//     Term 27 (APS4322-7000)/Term 28 (APS4322-5000)/FB Inputs/H{1..9 step 2} Z-Field <-> Data Pointer/HallSensorFieldsXYZ[{107..119 step 3}]  (5 links)
//     Term 27 (APS4322-7000)/Term 28 (APS4322-5000)/FB Inputs/I{0..8 step 2} X-Field <-> Data Pointer/HallSensorFieldsXYZ[{120..132 step 3}]  (5 links)
//     Term 27 (APS4322-7000)/Term 28 (APS4322-5000)/FB Inputs/I{0..8 step 2} Y-Field <-> Data Pointer/HallSensorFieldsXYZ[{121..133 step 3}]  (5 links)
//     Term 27 (APS4322-7000)/Term 28 (APS4322-5000)/FB Inputs/I{0..8 step 2} Z-Field <-> Data Pointer/HallSensorFieldsXYZ[{122..134 step 3}]  (5 links)
//     Term 27 (APS4322-7000)/Term 28 (APS4322-5000)/FB Inputs/J{1..9 step 2} X-Field <-> Data Pointer/HallSensorFieldsXYZ[{135..147 step 3}]  (5 links)
//     Term 27 (APS4322-7000)/Term 28 (APS4322-5000)/FB Inputs/J{1..9 step 2} Y-Field <-> Data Pointer/HallSensorFieldsXYZ[{136..148 step 3}]  (5 links)
//     Term 27 (APS4322-7000)/Term 28 (APS4322-5000)/FB Inputs/J{1..9 step 2} Z-Field <-> Data Pointer/HallSensorFieldsXYZ[{137..149 step 3}]  (5 links)
//     Term 27 (APS4322-7000)/Term 28 (APS4322-5000)/FB Inputs/Status <-> Data Pointer/FeedbackStatus
//   Device 3 (EtherCAT) <-> TcCOM Objects/XPlanar/Part1/APS4322_P1_3
//     Term 17 (APS4322-7000)/APS Comm Inputs/CommStatusWord <-> Data Pointer/MoverCommStatusWord
//     Term 17 (APS4322-7000)/APS Comm Inputs/Data {1..4} <-> Data Pointer/MoverCommDataIn[{0..3}]  (4 links)
//     Term 17 (APS4322-7000)/APS Comm Outputs/CommControlWord <-> Data Pointer/MoverCommControlWord
//     Term 17 (APS4322-7000)/APS Comm Outputs/Data 1 <-> Data Pointer/MoverCommDataOut
//     Term 17 (APS4322-7000)/APS Diagdata/DC Link Voltage <-> Data Pointer/DcLinkVoltage
//     Term 17 (APS4322-7000)/APS Diagdata/Power supply current <-> Data Pointer/PowerSupplyCurrent
//     Term 17 (APS4322-7000)/APS Inputs/StatusWord <-> Data Pointer/PowerUnitStatusWord
//     Term 17 (APS4322-7000)/APS Outputs/ControlWord <-> Data Pointer/PowerUnitControlWord
//     Term 17 (APS4322-7000)/APS Outputs/Current D 0X0 <-> Data Pointer/DCurrentSetPoints[0]
//     Term 17 (APS4322-7000)/APS Outputs/Current D 0X1 <-> Data Pointer/DCurrentSetPoints[1]
//     Term 17 (APS4322-7000)/APS Outputs/Current D 0X2 <-> Data Pointer/DCurrentSetPoints[2]
//     Term 17 (APS4322-7000)/APS Outputs/Current D 1X0 <-> Data Pointer/DCurrentSetPoints[6]
//     Term 17 (APS4322-7000)/APS Outputs/Current D 1X1 <-> Data Pointer/DCurrentSetPoints[7]
//     Term 17 (APS4322-7000)/APS Outputs/Current D 1X2 <-> Data Pointer/DCurrentSetPoints[8]
//     Term 17 (APS4322-7000)/APS Outputs/Current D 2X0 <-> Data Pointer/DCurrentSetPoints[12]
//     Term 17 (APS4322-7000)/APS Outputs/Current D 2X1 <-> Data Pointer/DCurrentSetPoints[13]
//     Term 17 (APS4322-7000)/APS Outputs/Current D 2X2 <-> Data Pointer/DCurrentSetPoints[14]
//     Term 17 (APS4322-7000)/APS Outputs/Current D 3X0 <-> Data Pointer/DCurrentSetPoints[18]
//     Term 17 (APS4322-7000)/APS Outputs/Current D 3X1 <-> Data Pointer/DCurrentSetPoints[19]
//     Term 17 (APS4322-7000)/APS Outputs/Current D 3X2 <-> Data Pointer/DCurrentSetPoints[20]
//     Term 17 (APS4322-7000)/APS Outputs/Current D 0Y0 <-> Data Pointer/DCurrentSetPoints[3]
//     Term 17 (APS4322-7000)/APS Outputs/Current D 0Y1 <-> Data Pointer/DCurrentSetPoints[4]
//     Term 17 (APS4322-7000)/APS Outputs/Current D 0Y2 <-> Data Pointer/DCurrentSetPoints[5]
//     Term 17 (APS4322-7000)/APS Outputs/Current D 1Y0 <-> Data Pointer/DCurrentSetPoints[9]
//     Term 17 (APS4322-7000)/APS Outputs/Current D 1Y1 <-> Data Pointer/DCurrentSetPoints[10]
//     Term 17 (APS4322-7000)/APS Outputs/Current D 1Y2 <-> Data Pointer/DCurrentSetPoints[11]
//     Term 17 (APS4322-7000)/APS Outputs/Current D 2Y0 <-> Data Pointer/DCurrentSetPoints[15]
//     Term 17 (APS4322-7000)/APS Outputs/Current D 2Y1 <-> Data Pointer/DCurrentSetPoints[16]
//     Term 17 (APS4322-7000)/APS Outputs/Current D 2Y2 <-> Data Pointer/DCurrentSetPoints[17]
//     Term 17 (APS4322-7000)/APS Outputs/Current D 3Y0 <-> Data Pointer/DCurrentSetPoints[21]
//     Term 17 (APS4322-7000)/APS Outputs/Current D 3Y1 <-> Data Pointer/DCurrentSetPoints[22]
//     Term 17 (APS4322-7000)/APS Outputs/Current D 3Y2 <-> Data Pointer/DCurrentSetPoints[23]
//     Term 17 (APS4322-7000)/APS Outputs/Current Q 0X0 <-> Data Pointer/QCurrentSetPoints[0]
//     Term 17 (APS4322-7000)/APS Outputs/Current Q 0X1 <-> Data Pointer/QCurrentSetPoints[1]
//     Term 17 (APS4322-7000)/APS Outputs/Current Q 0X2 <-> Data Pointer/QCurrentSetPoints[2]
//     Term 17 (APS4322-7000)/APS Outputs/Current Q 1X0 <-> Data Pointer/QCurrentSetPoints[6]
//     Term 17 (APS4322-7000)/APS Outputs/Current Q 1X1 <-> Data Pointer/QCurrentSetPoints[7]
//     Term 17 (APS4322-7000)/APS Outputs/Current Q 1X2 <-> Data Pointer/QCurrentSetPoints[8]
//     Term 17 (APS4322-7000)/APS Outputs/Current Q 2X0 <-> Data Pointer/QCurrentSetPoints[12]
//     Term 17 (APS4322-7000)/APS Outputs/Current Q 2X1 <-> Data Pointer/QCurrentSetPoints[13]
//     Term 17 (APS4322-7000)/APS Outputs/Current Q 2X2 <-> Data Pointer/QCurrentSetPoints[14]
//     Term 17 (APS4322-7000)/APS Outputs/Current Q 3X0 <-> Data Pointer/QCurrentSetPoints[18]
//     Term 17 (APS4322-7000)/APS Outputs/Current Q 3X1 <-> Data Pointer/QCurrentSetPoints[19]
//     Term 17 (APS4322-7000)/APS Outputs/Current Q 3X2 <-> Data Pointer/QCurrentSetPoints[20]
//     Term 17 (APS4322-7000)/APS Outputs/Current Q 0Y0 <-> Data Pointer/QCurrentSetPoints[3]
//     Term 17 (APS4322-7000)/APS Outputs/Current Q 0Y1 <-> Data Pointer/QCurrentSetPoints[4]
//     Term 17 (APS4322-7000)/APS Outputs/Current Q 0Y2 <-> Data Pointer/QCurrentSetPoints[5]
//     Term 17 (APS4322-7000)/APS Outputs/Current Q 1Y0 <-> Data Pointer/QCurrentSetPoints[9]
//     Term 17 (APS4322-7000)/APS Outputs/Current Q 1Y1 <-> Data Pointer/QCurrentSetPoints[10]
//     Term 17 (APS4322-7000)/APS Outputs/Current Q 1Y2 <-> Data Pointer/QCurrentSetPoints[11]
//     Term 17 (APS4322-7000)/APS Outputs/Current Q 2Y0 <-> Data Pointer/QCurrentSetPoints[15]
//     Term 17 (APS4322-7000)/APS Outputs/Current Q 2Y1 <-> Data Pointer/QCurrentSetPoints[16]
//     Term 17 (APS4322-7000)/APS Outputs/Current Q 2Y2 <-> Data Pointer/QCurrentSetPoints[17]
//     Term 17 (APS4322-7000)/APS Outputs/Current Q 3Y0 <-> Data Pointer/QCurrentSetPoints[21]
//     Term 17 (APS4322-7000)/APS Outputs/Current Q 3Y1 <-> Data Pointer/QCurrentSetPoints[22]
//     Term 17 (APS4322-7000)/APS Outputs/Current Q 3Y2 <-> Data Pointer/QCurrentSetPoints[23]
//     Term 17 (APS4322-7000)/APS Outputs/PhiE 0X0 <-> Data Pointer/PhiSetPoints[0]
//     Term 17 (APS4322-7000)/APS Outputs/PhiE 0X1 <-> Data Pointer/PhiSetPoints[1]
//     Term 17 (APS4322-7000)/APS Outputs/PhiE 0X2 <-> Data Pointer/PhiSetPoints[2]
//     Term 17 (APS4322-7000)/APS Outputs/PhiE 1X0 <-> Data Pointer/PhiSetPoints[6]
//     Term 17 (APS4322-7000)/APS Outputs/PhiE 1X1 <-> Data Pointer/PhiSetPoints[7]
//     Term 17 (APS4322-7000)/APS Outputs/PhiE 1X2 <-> Data Pointer/PhiSetPoints[8]
//     Term 17 (APS4322-7000)/APS Outputs/PhiE 2X0 <-> Data Pointer/PhiSetPoints[12]
//     Term 17 (APS4322-7000)/APS Outputs/PhiE 2X1 <-> Data Pointer/PhiSetPoints[13]
//     Term 17 (APS4322-7000)/APS Outputs/PhiE 2X2 <-> Data Pointer/PhiSetPoints[14]
//     Term 17 (APS4322-7000)/APS Outputs/PhiE 3X0 <-> Data Pointer/PhiSetPoints[18]
//     Term 17 (APS4322-7000)/APS Outputs/PhiE 3X1 <-> Data Pointer/PhiSetPoints[19]
//     Term 17 (APS4322-7000)/APS Outputs/PhiE 3X2 <-> Data Pointer/PhiSetPoints[20]
//     Term 17 (APS4322-7000)/APS Outputs/PhiE 0Y0 <-> Data Pointer/PhiSetPoints[3]
//     Term 17 (APS4322-7000)/APS Outputs/PhiE 0Y1 <-> Data Pointer/PhiSetPoints[4]
//     Term 17 (APS4322-7000)/APS Outputs/PhiE 0Y2 <-> Data Pointer/PhiSetPoints[5]
//     Term 17 (APS4322-7000)/APS Outputs/PhiE 1Y0 <-> Data Pointer/PhiSetPoints[9]
//     Term 17 (APS4322-7000)/APS Outputs/PhiE 1Y1 <-> Data Pointer/PhiSetPoints[10]
//     Term 17 (APS4322-7000)/APS Outputs/PhiE 1Y2 <-> Data Pointer/PhiSetPoints[11]
//     Term 17 (APS4322-7000)/APS Outputs/PhiE 2Y0 <-> Data Pointer/PhiSetPoints[15]
//     Term 17 (APS4322-7000)/APS Outputs/PhiE 2Y1 <-> Data Pointer/PhiSetPoints[16]
//     Term 17 (APS4322-7000)/APS Outputs/PhiE 2Y2 <-> Data Pointer/PhiSetPoints[17]
//     Term 17 (APS4322-7000)/APS Outputs/PhiE 3Y0 <-> Data Pointer/PhiSetPoints[21]
//     Term 17 (APS4322-7000)/APS Outputs/PhiE 3Y1 <-> Data Pointer/PhiSetPoints[22]
//     Term 17 (APS4322-7000)/APS Outputs/PhiE 3Y2 <-> Data Pointer/PhiSetPoints[23]
//     Term 17 (APS4322-7000)/Term 18 (APS4322-5000)/FB Inputs/A{0..8 step 2} X-Field <-> Data Pointer/HallSensorFieldsXYZ[{0..12 step 3}]  (5 links)
//     Term 17 (APS4322-7000)/Term 18 (APS4322-5000)/FB Inputs/A{0..8 step 2} Y-Field <-> Data Pointer/HallSensorFieldsXYZ[{1..13 step 3}]  (5 links)
//     Term 17 (APS4322-7000)/Term 18 (APS4322-5000)/FB Inputs/A{0..8 step 2} Z-Field <-> Data Pointer/HallSensorFieldsXYZ[{2..14 step 3}]  (5 links)
//     Term 17 (APS4322-7000)/Term 18 (APS4322-5000)/FB Inputs/B{1..9 step 2} X-Field <-> Data Pointer/HallSensorFieldsXYZ[{15..27 step 3}]  (5 links)
//     Term 17 (APS4322-7000)/Term 18 (APS4322-5000)/FB Inputs/B{1..9 step 2} Y-Field <-> Data Pointer/HallSensorFieldsXYZ[{16..28 step 3}]  (5 links)
//     Term 17 (APS4322-7000)/Term 18 (APS4322-5000)/FB Inputs/B{1..9 step 2} Z-Field <-> Data Pointer/HallSensorFieldsXYZ[{17..29 step 3}]  (5 links)
//     Term 17 (APS4322-7000)/Term 18 (APS4322-5000)/FB Inputs/C{0..8 step 2} X-Field <-> Data Pointer/HallSensorFieldsXYZ[{30..42 step 3}]  (5 links)
//     Term 17 (APS4322-7000)/Term 18 (APS4322-5000)/FB Inputs/C{0..8 step 2} Y-Field <-> Data Pointer/HallSensorFieldsXYZ[{31..43 step 3}]  (5 links)
//     Term 17 (APS4322-7000)/Term 18 (APS4322-5000)/FB Inputs/C{0..8 step 2} Z-Field <-> Data Pointer/HallSensorFieldsXYZ[{32..44 step 3}]  (5 links)
//     Term 17 (APS4322-7000)/Term 18 (APS4322-5000)/FB Inputs/D{1..9 step 2} X-Field <-> Data Pointer/HallSensorFieldsXYZ[{45..57 step 3}]  (5 links)
//     Term 17 (APS4322-7000)/Term 18 (APS4322-5000)/FB Inputs/D{1..9 step 2} Y-Field <-> Data Pointer/HallSensorFieldsXYZ[{46..58 step 3}]  (5 links)
//     Term 17 (APS4322-7000)/Term 18 (APS4322-5000)/FB Inputs/D{1..9 step 2} Z-Field <-> Data Pointer/HallSensorFieldsXYZ[{47..59 step 3}]  (5 links)
//     Term 17 (APS4322-7000)/Term 18 (APS4322-5000)/FB Inputs/E{0..8 step 2} X-Field <-> Data Pointer/HallSensorFieldsXYZ[{60..72 step 3}]  (5 links)
//     Term 17 (APS4322-7000)/Term 18 (APS4322-5000)/FB Inputs/E{0..8 step 2} Y-Field <-> Data Pointer/HallSensorFieldsXYZ[{61..73 step 3}]  (5 links)
//     Term 17 (APS4322-7000)/Term 18 (APS4322-5000)/FB Inputs/E{0..8 step 2} Z-Field <-> Data Pointer/HallSensorFieldsXYZ[{62..74 step 3}]  (5 links)
//     Term 17 (APS4322-7000)/Term 18 (APS4322-5000)/FB Inputs/F{1..9 step 2} X-Field <-> Data Pointer/HallSensorFieldsXYZ[{75..87 step 3}]  (5 links)
//     Term 17 (APS4322-7000)/Term 18 (APS4322-5000)/FB Inputs/F{1..9 step 2} Y-Field <-> Data Pointer/HallSensorFieldsXYZ[{76..88 step 3}]  (5 links)
//     Term 17 (APS4322-7000)/Term 18 (APS4322-5000)/FB Inputs/F{1..9 step 2} Z-Field <-> Data Pointer/HallSensorFieldsXYZ[{77..89 step 3}]  (5 links)
//     Term 17 (APS4322-7000)/Term 18 (APS4322-5000)/FB Inputs/G{0..8 step 2} X-Field <-> Data Pointer/HallSensorFieldsXYZ[{90..102 step 3}]  (5 links)
//     Term 17 (APS4322-7000)/Term 18 (APS4322-5000)/FB Inputs/G{0..8 step 2} Y-Field <-> Data Pointer/HallSensorFieldsXYZ[{91..103 step 3}]  (5 links)
//     Term 17 (APS4322-7000)/Term 18 (APS4322-5000)/FB Inputs/G{0..8 step 2} Z-Field <-> Data Pointer/HallSensorFieldsXYZ[{92..104 step 3}]  (5 links)
//     Term 17 (APS4322-7000)/Term 18 (APS4322-5000)/FB Inputs/H{1..9 step 2} X-Field <-> Data Pointer/HallSensorFieldsXYZ[{105..117 step 3}]  (5 links)
//     Term 17 (APS4322-7000)/Term 18 (APS4322-5000)/FB Inputs/H{1..9 step 2} Y-Field <-> Data Pointer/HallSensorFieldsXYZ[{106..118 step 3}]  (5 links)
//     Term 17 (APS4322-7000)/Term 18 (APS4322-5000)/FB Inputs/H{1..9 step 2} Z-Field <-> Data Pointer/HallSensorFieldsXYZ[{107..119 step 3}]  (5 links)
//     Term 17 (APS4322-7000)/Term 18 (APS4322-5000)/FB Inputs/I{0..8 step 2} X-Field <-> Data Pointer/HallSensorFieldsXYZ[{120..132 step 3}]  (5 links)
//     Term 17 (APS4322-7000)/Term 18 (APS4322-5000)/FB Inputs/I{0..8 step 2} Y-Field <-> Data Pointer/HallSensorFieldsXYZ[{121..133 step 3}]  (5 links)
//     Term 17 (APS4322-7000)/Term 18 (APS4322-5000)/FB Inputs/I{0..8 step 2} Z-Field <-> Data Pointer/HallSensorFieldsXYZ[{122..134 step 3}]  (5 links)
//     Term 17 (APS4322-7000)/Term 18 (APS4322-5000)/FB Inputs/J{1..9 step 2} X-Field <-> Data Pointer/HallSensorFieldsXYZ[{135..147 step 3}]  (5 links)
//     Term 17 (APS4322-7000)/Term 18 (APS4322-5000)/FB Inputs/J{1..9 step 2} Y-Field <-> Data Pointer/HallSensorFieldsXYZ[{136..148 step 3}]  (5 links)
//     Term 17 (APS4322-7000)/Term 18 (APS4322-5000)/FB Inputs/J{1..9 step 2} Z-Field <-> Data Pointer/HallSensorFieldsXYZ[{137..149 step 3}]  (5 links)
//     Term 17 (APS4322-7000)/Term 18 (APS4322-5000)/FB Inputs/Status <-> Data Pointer/FeedbackStatus
//   Device 3 (EtherCAT) <-> TcCOM Objects/XPlanar/Part1/APS4322_P1_4
//     Term 19 (APS4322-7000)/APS Comm Inputs/CommStatusWord <-> Data Pointer/MoverCommStatusWord
//     Term 19 (APS4322-7000)/APS Comm Inputs/Data {1..4} <-> Data Pointer/MoverCommDataIn[{0..3}]  (4 links)
//     Term 19 (APS4322-7000)/APS Comm Outputs/CommControlWord <-> Data Pointer/MoverCommControlWord
//     Term 19 (APS4322-7000)/APS Comm Outputs/Data 1 <-> Data Pointer/MoverCommDataOut
//     Term 19 (APS4322-7000)/APS Diagdata/DC Link Voltage <-> Data Pointer/DcLinkVoltage
//     Term 19 (APS4322-7000)/APS Diagdata/Power supply current <-> Data Pointer/PowerSupplyCurrent
//     Term 19 (APS4322-7000)/APS Inputs/StatusWord <-> Data Pointer/PowerUnitStatusWord
//     Term 19 (APS4322-7000)/APS Outputs/ControlWord <-> Data Pointer/PowerUnitControlWord
//     Term 19 (APS4322-7000)/APS Outputs/Current D 0X0 <-> Data Pointer/DCurrentSetPoints[0]
//     Term 19 (APS4322-7000)/APS Outputs/Current D 0X1 <-> Data Pointer/DCurrentSetPoints[1]
//     Term 19 (APS4322-7000)/APS Outputs/Current D 0X2 <-> Data Pointer/DCurrentSetPoints[2]
//     Term 19 (APS4322-7000)/APS Outputs/Current D 1X0 <-> Data Pointer/DCurrentSetPoints[6]
//     Term 19 (APS4322-7000)/APS Outputs/Current D 1X1 <-> Data Pointer/DCurrentSetPoints[7]
//     Term 19 (APS4322-7000)/APS Outputs/Current D 1X2 <-> Data Pointer/DCurrentSetPoints[8]
//     Term 19 (APS4322-7000)/APS Outputs/Current D 2X0 <-> Data Pointer/DCurrentSetPoints[12]
//     Term 19 (APS4322-7000)/APS Outputs/Current D 2X1 <-> Data Pointer/DCurrentSetPoints[13]
//     Term 19 (APS4322-7000)/APS Outputs/Current D 2X2 <-> Data Pointer/DCurrentSetPoints[14]
//     Term 19 (APS4322-7000)/APS Outputs/Current D 3X0 <-> Data Pointer/DCurrentSetPoints[18]
//     Term 19 (APS4322-7000)/APS Outputs/Current D 3X1 <-> Data Pointer/DCurrentSetPoints[19]
//     Term 19 (APS4322-7000)/APS Outputs/Current D 3X2 <-> Data Pointer/DCurrentSetPoints[20]
//     Term 19 (APS4322-7000)/APS Outputs/Current D 0Y0 <-> Data Pointer/DCurrentSetPoints[3]
//     Term 19 (APS4322-7000)/APS Outputs/Current D 0Y1 <-> Data Pointer/DCurrentSetPoints[4]
//     Term 19 (APS4322-7000)/APS Outputs/Current D 0Y2 <-> Data Pointer/DCurrentSetPoints[5]
//     Term 19 (APS4322-7000)/APS Outputs/Current D 1Y0 <-> Data Pointer/DCurrentSetPoints[9]
//     Term 19 (APS4322-7000)/APS Outputs/Current D 1Y1 <-> Data Pointer/DCurrentSetPoints[10]
//     Term 19 (APS4322-7000)/APS Outputs/Current D 1Y2 <-> Data Pointer/DCurrentSetPoints[11]
//     Term 19 (APS4322-7000)/APS Outputs/Current D 2Y0 <-> Data Pointer/DCurrentSetPoints[15]
//     Term 19 (APS4322-7000)/APS Outputs/Current D 2Y1 <-> Data Pointer/DCurrentSetPoints[16]
//     Term 19 (APS4322-7000)/APS Outputs/Current D 2Y2 <-> Data Pointer/DCurrentSetPoints[17]
//     Term 19 (APS4322-7000)/APS Outputs/Current D 3Y0 <-> Data Pointer/DCurrentSetPoints[21]
//     Term 19 (APS4322-7000)/APS Outputs/Current D 3Y1 <-> Data Pointer/DCurrentSetPoints[22]
//     Term 19 (APS4322-7000)/APS Outputs/Current D 3Y2 <-> Data Pointer/DCurrentSetPoints[23]
//     Term 19 (APS4322-7000)/APS Outputs/Current Q 0X0 <-> Data Pointer/QCurrentSetPoints[0]
//     Term 19 (APS4322-7000)/APS Outputs/Current Q 0X1 <-> Data Pointer/QCurrentSetPoints[1]
//     Term 19 (APS4322-7000)/APS Outputs/Current Q 0X2 <-> Data Pointer/QCurrentSetPoints[2]
//     Term 19 (APS4322-7000)/APS Outputs/Current Q 1X0 <-> Data Pointer/QCurrentSetPoints[6]
//     Term 19 (APS4322-7000)/APS Outputs/Current Q 1X1 <-> Data Pointer/QCurrentSetPoints[7]
//     Term 19 (APS4322-7000)/APS Outputs/Current Q 1X2 <-> Data Pointer/QCurrentSetPoints[8]
//     Term 19 (APS4322-7000)/APS Outputs/Current Q 2X0 <-> Data Pointer/QCurrentSetPoints[12]
//     Term 19 (APS4322-7000)/APS Outputs/Current Q 2X1 <-> Data Pointer/QCurrentSetPoints[13]
//     Term 19 (APS4322-7000)/APS Outputs/Current Q 2X2 <-> Data Pointer/QCurrentSetPoints[14]
//     Term 19 (APS4322-7000)/APS Outputs/Current Q 3X0 <-> Data Pointer/QCurrentSetPoints[18]
//     Term 19 (APS4322-7000)/APS Outputs/Current Q 3X1 <-> Data Pointer/QCurrentSetPoints[19]
//     Term 19 (APS4322-7000)/APS Outputs/Current Q 3X2 <-> Data Pointer/QCurrentSetPoints[20]
//     Term 19 (APS4322-7000)/APS Outputs/Current Q 0Y0 <-> Data Pointer/QCurrentSetPoints[3]
//     Term 19 (APS4322-7000)/APS Outputs/Current Q 0Y1 <-> Data Pointer/QCurrentSetPoints[4]
//     Term 19 (APS4322-7000)/APS Outputs/Current Q 0Y2 <-> Data Pointer/QCurrentSetPoints[5]
//     Term 19 (APS4322-7000)/APS Outputs/Current Q 1Y0 <-> Data Pointer/QCurrentSetPoints[9]
//     Term 19 (APS4322-7000)/APS Outputs/Current Q 1Y1 <-> Data Pointer/QCurrentSetPoints[10]
//     Term 19 (APS4322-7000)/APS Outputs/Current Q 1Y2 <-> Data Pointer/QCurrentSetPoints[11]
//     Term 19 (APS4322-7000)/APS Outputs/Current Q 2Y0 <-> Data Pointer/QCurrentSetPoints[15]
//     Term 19 (APS4322-7000)/APS Outputs/Current Q 2Y1 <-> Data Pointer/QCurrentSetPoints[16]
//     Term 19 (APS4322-7000)/APS Outputs/Current Q 2Y2 <-> Data Pointer/QCurrentSetPoints[17]
//     Term 19 (APS4322-7000)/APS Outputs/Current Q 3Y0 <-> Data Pointer/QCurrentSetPoints[21]
//     Term 19 (APS4322-7000)/APS Outputs/Current Q 3Y1 <-> Data Pointer/QCurrentSetPoints[22]
//     Term 19 (APS4322-7000)/APS Outputs/Current Q 3Y2 <-> Data Pointer/QCurrentSetPoints[23]
//     Term 19 (APS4322-7000)/APS Outputs/PhiE 0X0 <-> Data Pointer/PhiSetPoints[0]
//     Term 19 (APS4322-7000)/APS Outputs/PhiE 0X1 <-> Data Pointer/PhiSetPoints[1]
//     Term 19 (APS4322-7000)/APS Outputs/PhiE 0X2 <-> Data Pointer/PhiSetPoints[2]
//     Term 19 (APS4322-7000)/APS Outputs/PhiE 1X0 <-> Data Pointer/PhiSetPoints[6]
//     Term 19 (APS4322-7000)/APS Outputs/PhiE 1X1 <-> Data Pointer/PhiSetPoints[7]
//     Term 19 (APS4322-7000)/APS Outputs/PhiE 1X2 <-> Data Pointer/PhiSetPoints[8]
//     Term 19 (APS4322-7000)/APS Outputs/PhiE 2X0 <-> Data Pointer/PhiSetPoints[12]
//     Term 19 (APS4322-7000)/APS Outputs/PhiE 2X1 <-> Data Pointer/PhiSetPoints[13]
//     Term 19 (APS4322-7000)/APS Outputs/PhiE 2X2 <-> Data Pointer/PhiSetPoints[14]
//     Term 19 (APS4322-7000)/APS Outputs/PhiE 3X0 <-> Data Pointer/PhiSetPoints[18]
//     Term 19 (APS4322-7000)/APS Outputs/PhiE 3X1 <-> Data Pointer/PhiSetPoints[19]
//     Term 19 (APS4322-7000)/APS Outputs/PhiE 3X2 <-> Data Pointer/PhiSetPoints[20]
//     Term 19 (APS4322-7000)/APS Outputs/PhiE 0Y0 <-> Data Pointer/PhiSetPoints[3]
//     Term 19 (APS4322-7000)/APS Outputs/PhiE 0Y1 <-> Data Pointer/PhiSetPoints[4]
//     Term 19 (APS4322-7000)/APS Outputs/PhiE 0Y2 <-> Data Pointer/PhiSetPoints[5]
//     Term 19 (APS4322-7000)/APS Outputs/PhiE 1Y0 <-> Data Pointer/PhiSetPoints[9]
//     Term 19 (APS4322-7000)/APS Outputs/PhiE 1Y1 <-> Data Pointer/PhiSetPoints[10]
//     Term 19 (APS4322-7000)/APS Outputs/PhiE 1Y2 <-> Data Pointer/PhiSetPoints[11]
//     Term 19 (APS4322-7000)/APS Outputs/PhiE 2Y0 <-> Data Pointer/PhiSetPoints[15]
//     Term 19 (APS4322-7000)/APS Outputs/PhiE 2Y1 <-> Data Pointer/PhiSetPoints[16]
//     Term 19 (APS4322-7000)/APS Outputs/PhiE 2Y2 <-> Data Pointer/PhiSetPoints[17]
//     Term 19 (APS4322-7000)/APS Outputs/PhiE 3Y0 <-> Data Pointer/PhiSetPoints[21]
//     Term 19 (APS4322-7000)/APS Outputs/PhiE 3Y1 <-> Data Pointer/PhiSetPoints[22]
//     Term 19 (APS4322-7000)/APS Outputs/PhiE 3Y2 <-> Data Pointer/PhiSetPoints[23]
//     Term 19 (APS4322-7000)/Term 20 (APS4322-5000)/FB Inputs/A{0..8 step 2} X-Field <-> Data Pointer/HallSensorFieldsXYZ[{0..12 step 3}]  (5 links)
//     Term 19 (APS4322-7000)/Term 20 (APS4322-5000)/FB Inputs/A{0..8 step 2} Y-Field <-> Data Pointer/HallSensorFieldsXYZ[{1..13 step 3}]  (5 links)
//     Term 19 (APS4322-7000)/Term 20 (APS4322-5000)/FB Inputs/A{0..8 step 2} Z-Field <-> Data Pointer/HallSensorFieldsXYZ[{2..14 step 3}]  (5 links)
//     Term 19 (APS4322-7000)/Term 20 (APS4322-5000)/FB Inputs/B{1..9 step 2} X-Field <-> Data Pointer/HallSensorFieldsXYZ[{15..27 step 3}]  (5 links)
//     Term 19 (APS4322-7000)/Term 20 (APS4322-5000)/FB Inputs/B{1..9 step 2} Y-Field <-> Data Pointer/HallSensorFieldsXYZ[{16..28 step 3}]  (5 links)
//     Term 19 (APS4322-7000)/Term 20 (APS4322-5000)/FB Inputs/B{1..9 step 2} Z-Field <-> Data Pointer/HallSensorFieldsXYZ[{17..29 step 3}]  (5 links)
//     Term 19 (APS4322-7000)/Term 20 (APS4322-5000)/FB Inputs/C{0..8 step 2} X-Field <-> Data Pointer/HallSensorFieldsXYZ[{30..42 step 3}]  (5 links)
//     Term 19 (APS4322-7000)/Term 20 (APS4322-5000)/FB Inputs/C{0..8 step 2} Y-Field <-> Data Pointer/HallSensorFieldsXYZ[{31..43 step 3}]  (5 links)
//     Term 19 (APS4322-7000)/Term 20 (APS4322-5000)/FB Inputs/C{0..8 step 2} Z-Field <-> Data Pointer/HallSensorFieldsXYZ[{32..44 step 3}]  (5 links)
//     Term 19 (APS4322-7000)/Term 20 (APS4322-5000)/FB Inputs/D{1..9 step 2} X-Field <-> Data Pointer/HallSensorFieldsXYZ[{45..57 step 3}]  (5 links)
//     Term 19 (APS4322-7000)/Term 20 (APS4322-5000)/FB Inputs/D{1..9 step 2} Y-Field <-> Data Pointer/HallSensorFieldsXYZ[{46..58 step 3}]  (5 links)
//     Term 19 (APS4322-7000)/Term 20 (APS4322-5000)/FB Inputs/D{1..9 step 2} Z-Field <-> Data Pointer/HallSensorFieldsXYZ[{47..59 step 3}]  (5 links)
//     Term 19 (APS4322-7000)/Term 20 (APS4322-5000)/FB Inputs/E{0..8 step 2} X-Field <-> Data Pointer/HallSensorFieldsXYZ[{60..72 step 3}]  (5 links)
//     Term 19 (APS4322-7000)/Term 20 (APS4322-5000)/FB Inputs/E{0..8 step 2} Y-Field <-> Data Pointer/HallSensorFieldsXYZ[{61..73 step 3}]  (5 links)
//     Term 19 (APS4322-7000)/Term 20 (APS4322-5000)/FB Inputs/E{0..8 step 2} Z-Field <-> Data Pointer/HallSensorFieldsXYZ[{62..74 step 3}]  (5 links)
//     Term 19 (APS4322-7000)/Term 20 (APS4322-5000)/FB Inputs/F{1..9 step 2} X-Field <-> Data Pointer/HallSensorFieldsXYZ[{75..87 step 3}]  (5 links)
//     Term 19 (APS4322-7000)/Term 20 (APS4322-5000)/FB Inputs/F{1..9 step 2} Y-Field <-> Data Pointer/HallSensorFieldsXYZ[{76..88 step 3}]  (5 links)
//     Term 19 (APS4322-7000)/Term 20 (APS4322-5000)/FB Inputs/F{1..9 step 2} Z-Field <-> Data Pointer/HallSensorFieldsXYZ[{77..89 step 3}]  (5 links)
//     Term 19 (APS4322-7000)/Term 20 (APS4322-5000)/FB Inputs/G{0..8 step 2} X-Field <-> Data Pointer/HallSensorFieldsXYZ[{90..102 step 3}]  (5 links)
//     Term 19 (APS4322-7000)/Term 20 (APS4322-5000)/FB Inputs/G{0..8 step 2} Y-Field <-> Data Pointer/HallSensorFieldsXYZ[{91..103 step 3}]  (5 links)
//     Term 19 (APS4322-7000)/Term 20 (APS4322-5000)/FB Inputs/G{0..8 step 2} Z-Field <-> Data Pointer/HallSensorFieldsXYZ[{92..104 step 3}]  (5 links)
//     Term 19 (APS4322-7000)/Term 20 (APS4322-5000)/FB Inputs/H{1..9 step 2} X-Field <-> Data Pointer/HallSensorFieldsXYZ[{105..117 step 3}]  (5 links)
//     Term 19 (APS4322-7000)/Term 20 (APS4322-5000)/FB Inputs/H{1..9 step 2} Y-Field <-> Data Pointer/HallSensorFieldsXYZ[{106..118 step 3}]  (5 links)
//     Term 19 (APS4322-7000)/Term 20 (APS4322-5000)/FB Inputs/H{1..9 step 2} Z-Field <-> Data Pointer/HallSensorFieldsXYZ[{107..119 step 3}]  (5 links)
//     Term 19 (APS4322-7000)/Term 20 (APS4322-5000)/FB Inputs/I{0..8 step 2} X-Field <-> Data Pointer/HallSensorFieldsXYZ[{120..132 step 3}]  (5 links)
//     Term 19 (APS4322-7000)/Term 20 (APS4322-5000)/FB Inputs/I{0..8 step 2} Y-Field <-> Data Pointer/HallSensorFieldsXYZ[{121..133 step 3}]  (5 links)
//     Term 19 (APS4322-7000)/Term 20 (APS4322-5000)/FB Inputs/I{0..8 step 2} Z-Field <-> Data Pointer/HallSensorFieldsXYZ[{122..134 step 3}]  (5 links)
//     Term 19 (APS4322-7000)/Term 20 (APS4322-5000)/FB Inputs/J{1..9 step 2} X-Field <-> Data Pointer/HallSensorFieldsXYZ[{135..147 step 3}]  (5 links)
//     Term 19 (APS4322-7000)/Term 20 (APS4322-5000)/FB Inputs/J{1..9 step 2} Y-Field <-> Data Pointer/HallSensorFieldsXYZ[{136..148 step 3}]  (5 links)
//     Term 19 (APS4322-7000)/Term 20 (APS4322-5000)/FB Inputs/J{1..9 step 2} Z-Field <-> Data Pointer/HallSensorFieldsXYZ[{137..149 step 3}]  (5 links)
//     Term 19 (APS4322-7000)/Term 20 (APS4322-5000)/FB Inputs/Status <-> Data Pointer/FeedbackStatus
//   Device 3 (EtherCAT) <-> TcCOM Objects/XPlanar/Part1/APS4322_P1_7
//     Term 21 (APS4322-7000)/APS Comm Inputs/CommStatusWord <-> Data Pointer/MoverCommStatusWord
//     Term 21 (APS4322-7000)/APS Comm Inputs/Data {1..4} <-> Data Pointer/MoverCommDataIn[{0..3}]  (4 links)
//     Term 21 (APS4322-7000)/APS Comm Outputs/CommControlWord <-> Data Pointer/MoverCommControlWord
//     Term 21 (APS4322-7000)/APS Comm Outputs/Data 1 <-> Data Pointer/MoverCommDataOut
//     Term 21 (APS4322-7000)/APS Diagdata/DC Link Voltage <-> Data Pointer/DcLinkVoltage
//     Term 21 (APS4322-7000)/APS Diagdata/Power supply current <-> Data Pointer/PowerSupplyCurrent
//     Term 21 (APS4322-7000)/APS Inputs/StatusWord <-> Data Pointer/PowerUnitStatusWord
//     Term 21 (APS4322-7000)/APS Outputs/ControlWord <-> Data Pointer/PowerUnitControlWord
//     Term 21 (APS4322-7000)/APS Outputs/Current D 0X0 <-> Data Pointer/DCurrentSetPoints[0]
//     Term 21 (APS4322-7000)/APS Outputs/Current D 0X1 <-> Data Pointer/DCurrentSetPoints[1]
//     Term 21 (APS4322-7000)/APS Outputs/Current D 0X2 <-> Data Pointer/DCurrentSetPoints[2]
//     Term 21 (APS4322-7000)/APS Outputs/Current D 1X0 <-> Data Pointer/DCurrentSetPoints[6]
//     Term 21 (APS4322-7000)/APS Outputs/Current D 1X1 <-> Data Pointer/DCurrentSetPoints[7]
//     Term 21 (APS4322-7000)/APS Outputs/Current D 1X2 <-> Data Pointer/DCurrentSetPoints[8]
//     Term 21 (APS4322-7000)/APS Outputs/Current D 2X0 <-> Data Pointer/DCurrentSetPoints[12]
//     Term 21 (APS4322-7000)/APS Outputs/Current D 2X1 <-> Data Pointer/DCurrentSetPoints[13]
//     Term 21 (APS4322-7000)/APS Outputs/Current D 2X2 <-> Data Pointer/DCurrentSetPoints[14]
//     Term 21 (APS4322-7000)/APS Outputs/Current D 3X0 <-> Data Pointer/DCurrentSetPoints[18]
//     Term 21 (APS4322-7000)/APS Outputs/Current D 3X1 <-> Data Pointer/DCurrentSetPoints[19]
//     Term 21 (APS4322-7000)/APS Outputs/Current D 3X2 <-> Data Pointer/DCurrentSetPoints[20]
//     Term 21 (APS4322-7000)/APS Outputs/Current D 0Y0 <-> Data Pointer/DCurrentSetPoints[3]
//     Term 21 (APS4322-7000)/APS Outputs/Current D 0Y1 <-> Data Pointer/DCurrentSetPoints[4]
//     Term 21 (APS4322-7000)/APS Outputs/Current D 0Y2 <-> Data Pointer/DCurrentSetPoints[5]
//     Term 21 (APS4322-7000)/APS Outputs/Current D 1Y0 <-> Data Pointer/DCurrentSetPoints[9]
//     Term 21 (APS4322-7000)/APS Outputs/Current D 1Y1 <-> Data Pointer/DCurrentSetPoints[10]
//     Term 21 (APS4322-7000)/APS Outputs/Current D 1Y2 <-> Data Pointer/DCurrentSetPoints[11]
//     Term 21 (APS4322-7000)/APS Outputs/Current D 2Y0 <-> Data Pointer/DCurrentSetPoints[15]
//     Term 21 (APS4322-7000)/APS Outputs/Current D 2Y1 <-> Data Pointer/DCurrentSetPoints[16]
//     Term 21 (APS4322-7000)/APS Outputs/Current D 2Y2 <-> Data Pointer/DCurrentSetPoints[17]
//     Term 21 (APS4322-7000)/APS Outputs/Current D 3Y0 <-> Data Pointer/DCurrentSetPoints[21]
//     Term 21 (APS4322-7000)/APS Outputs/Current D 3Y1 <-> Data Pointer/DCurrentSetPoints[22]
//     Term 21 (APS4322-7000)/APS Outputs/Current D 3Y2 <-> Data Pointer/DCurrentSetPoints[23]
//     Term 21 (APS4322-7000)/APS Outputs/Current Q 0X0 <-> Data Pointer/QCurrentSetPoints[0]
//     Term 21 (APS4322-7000)/APS Outputs/Current Q 0X1 <-> Data Pointer/QCurrentSetPoints[1]
//     Term 21 (APS4322-7000)/APS Outputs/Current Q 0X2 <-> Data Pointer/QCurrentSetPoints[2]
//     Term 21 (APS4322-7000)/APS Outputs/Current Q 1X0 <-> Data Pointer/QCurrentSetPoints[6]
//     Term 21 (APS4322-7000)/APS Outputs/Current Q 1X1 <-> Data Pointer/QCurrentSetPoints[7]
//     Term 21 (APS4322-7000)/APS Outputs/Current Q 1X2 <-> Data Pointer/QCurrentSetPoints[8]
//     Term 21 (APS4322-7000)/APS Outputs/Current Q 2X0 <-> Data Pointer/QCurrentSetPoints[12]
//     Term 21 (APS4322-7000)/APS Outputs/Current Q 2X1 <-> Data Pointer/QCurrentSetPoints[13]
//     Term 21 (APS4322-7000)/APS Outputs/Current Q 2X2 <-> Data Pointer/QCurrentSetPoints[14]
//     Term 21 (APS4322-7000)/APS Outputs/Current Q 3X0 <-> Data Pointer/QCurrentSetPoints[18]
//     Term 21 (APS4322-7000)/APS Outputs/Current Q 3X1 <-> Data Pointer/QCurrentSetPoints[19]
//     Term 21 (APS4322-7000)/APS Outputs/Current Q 3X2 <-> Data Pointer/QCurrentSetPoints[20]
//     Term 21 (APS4322-7000)/APS Outputs/Current Q 0Y0 <-> Data Pointer/QCurrentSetPoints[3]
//     Term 21 (APS4322-7000)/APS Outputs/Current Q 0Y1 <-> Data Pointer/QCurrentSetPoints[4]
//     Term 21 (APS4322-7000)/APS Outputs/Current Q 0Y2 <-> Data Pointer/QCurrentSetPoints[5]
//     Term 21 (APS4322-7000)/APS Outputs/Current Q 1Y0 <-> Data Pointer/QCurrentSetPoints[9]
//     Term 21 (APS4322-7000)/APS Outputs/Current Q 1Y1 <-> Data Pointer/QCurrentSetPoints[10]
//     Term 21 (APS4322-7000)/APS Outputs/Current Q 1Y2 <-> Data Pointer/QCurrentSetPoints[11]
//     Term 21 (APS4322-7000)/APS Outputs/Current Q 2Y0 <-> Data Pointer/QCurrentSetPoints[15]
//     Term 21 (APS4322-7000)/APS Outputs/Current Q 2Y1 <-> Data Pointer/QCurrentSetPoints[16]
//     Term 21 (APS4322-7000)/APS Outputs/Current Q 2Y2 <-> Data Pointer/QCurrentSetPoints[17]
//     Term 21 (APS4322-7000)/APS Outputs/Current Q 3Y0 <-> Data Pointer/QCurrentSetPoints[21]
//     Term 21 (APS4322-7000)/APS Outputs/Current Q 3Y1 <-> Data Pointer/QCurrentSetPoints[22]
//     Term 21 (APS4322-7000)/APS Outputs/Current Q 3Y2 <-> Data Pointer/QCurrentSetPoints[23]
//     Term 21 (APS4322-7000)/APS Outputs/PhiE 0X0 <-> Data Pointer/PhiSetPoints[0]
//     Term 21 (APS4322-7000)/APS Outputs/PhiE 0X1 <-> Data Pointer/PhiSetPoints[1]
//     Term 21 (APS4322-7000)/APS Outputs/PhiE 0X2 <-> Data Pointer/PhiSetPoints[2]
//     Term 21 (APS4322-7000)/APS Outputs/PhiE 1X0 <-> Data Pointer/PhiSetPoints[6]
//     Term 21 (APS4322-7000)/APS Outputs/PhiE 1X1 <-> Data Pointer/PhiSetPoints[7]
//     Term 21 (APS4322-7000)/APS Outputs/PhiE 1X2 <-> Data Pointer/PhiSetPoints[8]
//     Term 21 (APS4322-7000)/APS Outputs/PhiE 2X0 <-> Data Pointer/PhiSetPoints[12]
//     Term 21 (APS4322-7000)/APS Outputs/PhiE 2X1 <-> Data Pointer/PhiSetPoints[13]
//     Term 21 (APS4322-7000)/APS Outputs/PhiE 2X2 <-> Data Pointer/PhiSetPoints[14]
//     Term 21 (APS4322-7000)/APS Outputs/PhiE 3X0 <-> Data Pointer/PhiSetPoints[18]
//     Term 21 (APS4322-7000)/APS Outputs/PhiE 3X1 <-> Data Pointer/PhiSetPoints[19]
//     Term 21 (APS4322-7000)/APS Outputs/PhiE 3X2 <-> Data Pointer/PhiSetPoints[20]
//     Term 21 (APS4322-7000)/APS Outputs/PhiE 0Y0 <-> Data Pointer/PhiSetPoints[3]
//     Term 21 (APS4322-7000)/APS Outputs/PhiE 0Y1 <-> Data Pointer/PhiSetPoints[4]
//     Term 21 (APS4322-7000)/APS Outputs/PhiE 0Y2 <-> Data Pointer/PhiSetPoints[5]
//     Term 21 (APS4322-7000)/APS Outputs/PhiE 1Y0 <-> Data Pointer/PhiSetPoints[9]
//     Term 21 (APS4322-7000)/APS Outputs/PhiE 1Y1 <-> Data Pointer/PhiSetPoints[10]
//     Term 21 (APS4322-7000)/APS Outputs/PhiE 1Y2 <-> Data Pointer/PhiSetPoints[11]
//     Term 21 (APS4322-7000)/APS Outputs/PhiE 2Y0 <-> Data Pointer/PhiSetPoints[15]
//     Term 21 (APS4322-7000)/APS Outputs/PhiE 2Y1 <-> Data Pointer/PhiSetPoints[16]
//     Term 21 (APS4322-7000)/APS Outputs/PhiE 2Y2 <-> Data Pointer/PhiSetPoints[17]
//     Term 21 (APS4322-7000)/APS Outputs/PhiE 3Y0 <-> Data Pointer/PhiSetPoints[21]
//     Term 21 (APS4322-7000)/APS Outputs/PhiE 3Y1 <-> Data Pointer/PhiSetPoints[22]
//     Term 21 (APS4322-7000)/APS Outputs/PhiE 3Y2 <-> Data Pointer/PhiSetPoints[23]
//     Term 21 (APS4322-7000)/Term 22 (APS4322-5000)/FB Inputs/A{0..8 step 2} X-Field <-> Data Pointer/HallSensorFieldsXYZ[{0..12 step 3}]  (5 links)
//     Term 21 (APS4322-7000)/Term 22 (APS4322-5000)/FB Inputs/A{0..8 step 2} Y-Field <-> Data Pointer/HallSensorFieldsXYZ[{1..13 step 3}]  (5 links)
//     Term 21 (APS4322-7000)/Term 22 (APS4322-5000)/FB Inputs/A{0..8 step 2} Z-Field <-> Data Pointer/HallSensorFieldsXYZ[{2..14 step 3}]  (5 links)
//     Term 21 (APS4322-7000)/Term 22 (APS4322-5000)/FB Inputs/B{1..9 step 2} X-Field <-> Data Pointer/HallSensorFieldsXYZ[{15..27 step 3}]  (5 links)
//     Term 21 (APS4322-7000)/Term 22 (APS4322-5000)/FB Inputs/B{1..9 step 2} Y-Field <-> Data Pointer/HallSensorFieldsXYZ[{16..28 step 3}]  (5 links)
//     Term 21 (APS4322-7000)/Term 22 (APS4322-5000)/FB Inputs/B{1..9 step 2} Z-Field <-> Data Pointer/HallSensorFieldsXYZ[{17..29 step 3}]  (5 links)
//     Term 21 (APS4322-7000)/Term 22 (APS4322-5000)/FB Inputs/C{0..8 step 2} X-Field <-> Data Pointer/HallSensorFieldsXYZ[{30..42 step 3}]  (5 links)
//     Term 21 (APS4322-7000)/Term 22 (APS4322-5000)/FB Inputs/C{0..8 step 2} Y-Field <-> Data Pointer/HallSensorFieldsXYZ[{31..43 step 3}]  (5 links)
//     Term 21 (APS4322-7000)/Term 22 (APS4322-5000)/FB Inputs/C{0..8 step 2} Z-Field <-> Data Pointer/HallSensorFieldsXYZ[{32..44 step 3}]  (5 links)
//     Term 21 (APS4322-7000)/Term 22 (APS4322-5000)/FB Inputs/D{1..9 step 2} X-Field <-> Data Pointer/HallSensorFieldsXYZ[{45..57 step 3}]  (5 links)
//     Term 21 (APS4322-7000)/Term 22 (APS4322-5000)/FB Inputs/D{1..9 step 2} Y-Field <-> Data Pointer/HallSensorFieldsXYZ[{46..58 step 3}]  (5 links)
//     Term 21 (APS4322-7000)/Term 22 (APS4322-5000)/FB Inputs/D{1..9 step 2} Z-Field <-> Data Pointer/HallSensorFieldsXYZ[{47..59 step 3}]  (5 links)
//     Term 21 (APS4322-7000)/Term 22 (APS4322-5000)/FB Inputs/E{0..8 step 2} X-Field <-> Data Pointer/HallSensorFieldsXYZ[{60..72 step 3}]  (5 links)
//     Term 21 (APS4322-7000)/Term 22 (APS4322-5000)/FB Inputs/E{0..8 step 2} Y-Field <-> Data Pointer/HallSensorFieldsXYZ[{61..73 step 3}]  (5 links)
//     Term 21 (APS4322-7000)/Term 22 (APS4322-5000)/FB Inputs/E{0..8 step 2} Z-Field <-> Data Pointer/HallSensorFieldsXYZ[{62..74 step 3}]  (5 links)
//     Term 21 (APS4322-7000)/Term 22 (APS4322-5000)/FB Inputs/F{1..9 step 2} X-Field <-> Data Pointer/HallSensorFieldsXYZ[{75..87 step 3}]  (5 links)
//     Term 21 (APS4322-7000)/Term 22 (APS4322-5000)/FB Inputs/F{1..9 step 2} Y-Field <-> Data Pointer/HallSensorFieldsXYZ[{76..88 step 3}]  (5 links)
//     Term 21 (APS4322-7000)/Term 22 (APS4322-5000)/FB Inputs/F{1..9 step 2} Z-Field <-> Data Pointer/HallSensorFieldsXYZ[{77..89 step 3}]  (5 links)
//     Term 21 (APS4322-7000)/Term 22 (APS4322-5000)/FB Inputs/G{0..8 step 2} X-Field <-> Data Pointer/HallSensorFieldsXYZ[{90..102 step 3}]  (5 links)
//     Term 21 (APS4322-7000)/Term 22 (APS4322-5000)/FB Inputs/G{0..8 step 2} Y-Field <-> Data Pointer/HallSensorFieldsXYZ[{91..103 step 3}]  (5 links)
//     Term 21 (APS4322-7000)/Term 22 (APS4322-5000)/FB Inputs/G{0..8 step 2} Z-Field <-> Data Pointer/HallSensorFieldsXYZ[{92..104 step 3}]  (5 links)
//     Term 21 (APS4322-7000)/Term 22 (APS4322-5000)/FB Inputs/H{1..9 step 2} X-Field <-> Data Pointer/HallSensorFieldsXYZ[{105..117 step 3}]  (5 links)
//     Term 21 (APS4322-7000)/Term 22 (APS4322-5000)/FB Inputs/H{1..9 step 2} Y-Field <-> Data Pointer/HallSensorFieldsXYZ[{106..118 step 3}]  (5 links)
//     Term 21 (APS4322-7000)/Term 22 (APS4322-5000)/FB Inputs/H{1..9 step 2} Z-Field <-> Data Pointer/HallSensorFieldsXYZ[{107..119 step 3}]  (5 links)
//     Term 21 (APS4322-7000)/Term 22 (APS4322-5000)/FB Inputs/I{0..8 step 2} X-Field <-> Data Pointer/HallSensorFieldsXYZ[{120..132 step 3}]  (5 links)
//     Term 21 (APS4322-7000)/Term 22 (APS4322-5000)/FB Inputs/I{0..8 step 2} Y-Field <-> Data Pointer/HallSensorFieldsXYZ[{121..133 step 3}]  (5 links)
//     Term 21 (APS4322-7000)/Term 22 (APS4322-5000)/FB Inputs/I{0..8 step 2} Z-Field <-> Data Pointer/HallSensorFieldsXYZ[{122..134 step 3}]  (5 links)
//     Term 21 (APS4322-7000)/Term 22 (APS4322-5000)/FB Inputs/J{1..9 step 2} X-Field <-> Data Pointer/HallSensorFieldsXYZ[{135..147 step 3}]  (5 links)
//     Term 21 (APS4322-7000)/Term 22 (APS4322-5000)/FB Inputs/J{1..9 step 2} Y-Field <-> Data Pointer/HallSensorFieldsXYZ[{136..148 step 3}]  (5 links)
//     Term 21 (APS4322-7000)/Term 22 (APS4322-5000)/FB Inputs/J{1..9 step 2} Z-Field <-> Data Pointer/HallSensorFieldsXYZ[{137..149 step 3}]  (5 links)
//     Term 21 (APS4322-7000)/Term 22 (APS4322-5000)/FB Inputs/Status <-> Data Pointer/FeedbackStatus
//   Device 3 (EtherCAT) <-> TcCOM Objects/XPlanar/Part1/APS4322_P1_8
//     Term 23 (APS4322-7000)/APS Comm Inputs/CommStatusWord <-> Data Pointer/MoverCommStatusWord
//     Term 23 (APS4322-7000)/APS Comm Inputs/Data {1..4} <-> Data Pointer/MoverCommDataIn[{0..3}]  (4 links)
//     Term 23 (APS4322-7000)/APS Comm Outputs/CommControlWord <-> Data Pointer/MoverCommControlWord
//     Term 23 (APS4322-7000)/APS Comm Outputs/Data 1 <-> Data Pointer/MoverCommDataOut
//     Term 23 (APS4322-7000)/APS Diagdata/DC Link Voltage <-> Data Pointer/DcLinkVoltage
//     Term 23 (APS4322-7000)/APS Diagdata/Power supply current <-> Data Pointer/PowerSupplyCurrent
//     Term 23 (APS4322-7000)/APS Inputs/StatusWord <-> Data Pointer/PowerUnitStatusWord
//     Term 23 (APS4322-7000)/APS Outputs/ControlWord <-> Data Pointer/PowerUnitControlWord
//     Term 23 (APS4322-7000)/APS Outputs/Current D 0X0 <-> Data Pointer/DCurrentSetPoints[0]
//     Term 23 (APS4322-7000)/APS Outputs/Current D 0X1 <-> Data Pointer/DCurrentSetPoints[1]
//     Term 23 (APS4322-7000)/APS Outputs/Current D 0X2 <-> Data Pointer/DCurrentSetPoints[2]
//     Term 23 (APS4322-7000)/APS Outputs/Current D 1X0 <-> Data Pointer/DCurrentSetPoints[6]
//     Term 23 (APS4322-7000)/APS Outputs/Current D 1X1 <-> Data Pointer/DCurrentSetPoints[7]
//     Term 23 (APS4322-7000)/APS Outputs/Current D 1X2 <-> Data Pointer/DCurrentSetPoints[8]
//     Term 23 (APS4322-7000)/APS Outputs/Current D 2X0 <-> Data Pointer/DCurrentSetPoints[12]
//     Term 23 (APS4322-7000)/APS Outputs/Current D 2X1 <-> Data Pointer/DCurrentSetPoints[13]
//     Term 23 (APS4322-7000)/APS Outputs/Current D 2X2 <-> Data Pointer/DCurrentSetPoints[14]
//     Term 23 (APS4322-7000)/APS Outputs/Current D 3X0 <-> Data Pointer/DCurrentSetPoints[18]
//     Term 23 (APS4322-7000)/APS Outputs/Current D 3X1 <-> Data Pointer/DCurrentSetPoints[19]
//     Term 23 (APS4322-7000)/APS Outputs/Current D 3X2 <-> Data Pointer/DCurrentSetPoints[20]
//     Term 23 (APS4322-7000)/APS Outputs/Current D 0Y0 <-> Data Pointer/DCurrentSetPoints[3]
//     Term 23 (APS4322-7000)/APS Outputs/Current D 0Y1 <-> Data Pointer/DCurrentSetPoints[4]
//     Term 23 (APS4322-7000)/APS Outputs/Current D 0Y2 <-> Data Pointer/DCurrentSetPoints[5]
//     Term 23 (APS4322-7000)/APS Outputs/Current D 1Y0 <-> Data Pointer/DCurrentSetPoints[9]
//     Term 23 (APS4322-7000)/APS Outputs/Current D 1Y1 <-> Data Pointer/DCurrentSetPoints[10]
//     Term 23 (APS4322-7000)/APS Outputs/Current D 1Y2 <-> Data Pointer/DCurrentSetPoints[11]
//     Term 23 (APS4322-7000)/APS Outputs/Current D 2Y0 <-> Data Pointer/DCurrentSetPoints[15]
//     Term 23 (APS4322-7000)/APS Outputs/Current D 2Y1 <-> Data Pointer/DCurrentSetPoints[16]
//     Term 23 (APS4322-7000)/APS Outputs/Current D 2Y2 <-> Data Pointer/DCurrentSetPoints[17]
//     Term 23 (APS4322-7000)/APS Outputs/Current D 3Y0 <-> Data Pointer/DCurrentSetPoints[21]
//     Term 23 (APS4322-7000)/APS Outputs/Current D 3Y1 <-> Data Pointer/DCurrentSetPoints[22]
//     Term 23 (APS4322-7000)/APS Outputs/Current D 3Y2 <-> Data Pointer/DCurrentSetPoints[23]
//     Term 23 (APS4322-7000)/APS Outputs/Current Q 0X0 <-> Data Pointer/QCurrentSetPoints[0]
//     Term 23 (APS4322-7000)/APS Outputs/Current Q 0X1 <-> Data Pointer/QCurrentSetPoints[1]
//     Term 23 (APS4322-7000)/APS Outputs/Current Q 0X2 <-> Data Pointer/QCurrentSetPoints[2]
//     Term 23 (APS4322-7000)/APS Outputs/Current Q 1X0 <-> Data Pointer/QCurrentSetPoints[6]
//     Term 23 (APS4322-7000)/APS Outputs/Current Q 1X1 <-> Data Pointer/QCurrentSetPoints[7]
//     Term 23 (APS4322-7000)/APS Outputs/Current Q 1X2 <-> Data Pointer/QCurrentSetPoints[8]
//     Term 23 (APS4322-7000)/APS Outputs/Current Q 2X0 <-> Data Pointer/QCurrentSetPoints[12]
//     Term 23 (APS4322-7000)/APS Outputs/Current Q 2X1 <-> Data Pointer/QCurrentSetPoints[13]
//     Term 23 (APS4322-7000)/APS Outputs/Current Q 2X2 <-> Data Pointer/QCurrentSetPoints[14]
//     Term 23 (APS4322-7000)/APS Outputs/Current Q 3X0 <-> Data Pointer/QCurrentSetPoints[18]
//     Term 23 (APS4322-7000)/APS Outputs/Current Q 3X1 <-> Data Pointer/QCurrentSetPoints[19]
//     Term 23 (APS4322-7000)/APS Outputs/Current Q 3X2 <-> Data Pointer/QCurrentSetPoints[20]
//     Term 23 (APS4322-7000)/APS Outputs/Current Q 0Y0 <-> Data Pointer/QCurrentSetPoints[3]
//     Term 23 (APS4322-7000)/APS Outputs/Current Q 0Y1 <-> Data Pointer/QCurrentSetPoints[4]
//     Term 23 (APS4322-7000)/APS Outputs/Current Q 0Y2 <-> Data Pointer/QCurrentSetPoints[5]
//     Term 23 (APS4322-7000)/APS Outputs/Current Q 1Y0 <-> Data Pointer/QCurrentSetPoints[9]
//     Term 23 (APS4322-7000)/APS Outputs/Current Q 1Y1 <-> Data Pointer/QCurrentSetPoints[10]
//     Term 23 (APS4322-7000)/APS Outputs/Current Q 1Y2 <-> Data Pointer/QCurrentSetPoints[11]
//     Term 23 (APS4322-7000)/APS Outputs/Current Q 2Y0 <-> Data Pointer/QCurrentSetPoints[15]
//     Term 23 (APS4322-7000)/APS Outputs/Current Q 2Y1 <-> Data Pointer/QCurrentSetPoints[16]
//     Term 23 (APS4322-7000)/APS Outputs/Current Q 2Y2 <-> Data Pointer/QCurrentSetPoints[17]
//     Term 23 (APS4322-7000)/APS Outputs/Current Q 3Y0 <-> Data Pointer/QCurrentSetPoints[21]
//     Term 23 (APS4322-7000)/APS Outputs/Current Q 3Y1 <-> Data Pointer/QCurrentSetPoints[22]
//     Term 23 (APS4322-7000)/APS Outputs/Current Q 3Y2 <-> Data Pointer/QCurrentSetPoints[23]
//     Term 23 (APS4322-7000)/APS Outputs/PhiE 0X0 <-> Data Pointer/PhiSetPoints[0]
//     Term 23 (APS4322-7000)/APS Outputs/PhiE 0X1 <-> Data Pointer/PhiSetPoints[1]
//     Term 23 (APS4322-7000)/APS Outputs/PhiE 0X2 <-> Data Pointer/PhiSetPoints[2]
//     Term 23 (APS4322-7000)/APS Outputs/PhiE 1X0 <-> Data Pointer/PhiSetPoints[6]
//     Term 23 (APS4322-7000)/APS Outputs/PhiE 1X1 <-> Data Pointer/PhiSetPoints[7]
//     Term 23 (APS4322-7000)/APS Outputs/PhiE 1X2 <-> Data Pointer/PhiSetPoints[8]
//     Term 23 (APS4322-7000)/APS Outputs/PhiE 2X0 <-> Data Pointer/PhiSetPoints[12]
//     Term 23 (APS4322-7000)/APS Outputs/PhiE 2X1 <-> Data Pointer/PhiSetPoints[13]
//     Term 23 (APS4322-7000)/APS Outputs/PhiE 2X2 <-> Data Pointer/PhiSetPoints[14]
//     Term 23 (APS4322-7000)/APS Outputs/PhiE 3X0 <-> Data Pointer/PhiSetPoints[18]
//     Term 23 (APS4322-7000)/APS Outputs/PhiE 3X1 <-> Data Pointer/PhiSetPoints[19]
//     Term 23 (APS4322-7000)/APS Outputs/PhiE 3X2 <-> Data Pointer/PhiSetPoints[20]
//     Term 23 (APS4322-7000)/APS Outputs/PhiE 0Y0 <-> Data Pointer/PhiSetPoints[3]
//     Term 23 (APS4322-7000)/APS Outputs/PhiE 0Y1 <-> Data Pointer/PhiSetPoints[4]
//     Term 23 (APS4322-7000)/APS Outputs/PhiE 0Y2 <-> Data Pointer/PhiSetPoints[5]
//     Term 23 (APS4322-7000)/APS Outputs/PhiE 1Y0 <-> Data Pointer/PhiSetPoints[9]
//     Term 23 (APS4322-7000)/APS Outputs/PhiE 1Y1 <-> Data Pointer/PhiSetPoints[10]
//     Term 23 (APS4322-7000)/APS Outputs/PhiE 1Y2 <-> Data Pointer/PhiSetPoints[11]
//     Term 23 (APS4322-7000)/APS Outputs/PhiE 2Y0 <-> Data Pointer/PhiSetPoints[15]
//     Term 23 (APS4322-7000)/APS Outputs/PhiE 2Y1 <-> Data Pointer/PhiSetPoints[16]
//     Term 23 (APS4322-7000)/APS Outputs/PhiE 2Y2 <-> Data Pointer/PhiSetPoints[17]
//     Term 23 (APS4322-7000)/APS Outputs/PhiE 3Y0 <-> Data Pointer/PhiSetPoints[21]
//     Term 23 (APS4322-7000)/APS Outputs/PhiE 3Y1 <-> Data Pointer/PhiSetPoints[22]
//     Term 23 (APS4322-7000)/APS Outputs/PhiE 3Y2 <-> Data Pointer/PhiSetPoints[23]
//     Term 23 (APS4322-7000)/Term 24 (APS4322-5000)/FB Inputs/A{0..8 step 2} X-Field <-> Data Pointer/HallSensorFieldsXYZ[{0..12 step 3}]  (5 links)
//     Term 23 (APS4322-7000)/Term 24 (APS4322-5000)/FB Inputs/A{0..8 step 2} Y-Field <-> Data Pointer/HallSensorFieldsXYZ[{1..13 step 3}]  (5 links)
//     Term 23 (APS4322-7000)/Term 24 (APS4322-5000)/FB Inputs/A{0..8 step 2} Z-Field <-> Data Pointer/HallSensorFieldsXYZ[{2..14 step 3}]  (5 links)
//     Term 23 (APS4322-7000)/Term 24 (APS4322-5000)/FB Inputs/B{1..9 step 2} X-Field <-> Data Pointer/HallSensorFieldsXYZ[{15..27 step 3}]  (5 links)
//     Term 23 (APS4322-7000)/Term 24 (APS4322-5000)/FB Inputs/B{1..9 step 2} Y-Field <-> Data Pointer/HallSensorFieldsXYZ[{16..28 step 3}]  (5 links)
//     Term 23 (APS4322-7000)/Term 24 (APS4322-5000)/FB Inputs/B{1..9 step 2} Z-Field <-> Data Pointer/HallSensorFieldsXYZ[{17..29 step 3}]  (5 links)
//     Term 23 (APS4322-7000)/Term 24 (APS4322-5000)/FB Inputs/C{0..8 step 2} X-Field <-> Data Pointer/HallSensorFieldsXYZ[{30..42 step 3}]  (5 links)
//     Term 23 (APS4322-7000)/Term 24 (APS4322-5000)/FB Inputs/C{0..8 step 2} Y-Field <-> Data Pointer/HallSensorFieldsXYZ[{31..43 step 3}]  (5 links)
//     Term 23 (APS4322-7000)/Term 24 (APS4322-5000)/FB Inputs/C{0..8 step 2} Z-Field <-> Data Pointer/HallSensorFieldsXYZ[{32..44 step 3}]  (5 links)
//     Term 23 (APS4322-7000)/Term 24 (APS4322-5000)/FB Inputs/D{1..9 step 2} X-Field <-> Data Pointer/HallSensorFieldsXYZ[{45..57 step 3}]  (5 links)
//     Term 23 (APS4322-7000)/Term 24 (APS4322-5000)/FB Inputs/D{1..9 step 2} Y-Field <-> Data Pointer/HallSensorFieldsXYZ[{46..58 step 3}]  (5 links)
//     Term 23 (APS4322-7000)/Term 24 (APS4322-5000)/FB Inputs/D{1..9 step 2} Z-Field <-> Data Pointer/HallSensorFieldsXYZ[{47..59 step 3}]  (5 links)
//     Term 23 (APS4322-7000)/Term 24 (APS4322-5000)/FB Inputs/E{0..8 step 2} X-Field <-> Data Pointer/HallSensorFieldsXYZ[{60..72 step 3}]  (5 links)
//     Term 23 (APS4322-7000)/Term 24 (APS4322-5000)/FB Inputs/E{0..8 step 2} Y-Field <-> Data Pointer/HallSensorFieldsXYZ[{61..73 step 3}]  (5 links)
//     Term 23 (APS4322-7000)/Term 24 (APS4322-5000)/FB Inputs/E{0..8 step 2} Z-Field <-> Data Pointer/HallSensorFieldsXYZ[{62..74 step 3}]  (5 links)
//     Term 23 (APS4322-7000)/Term 24 (APS4322-5000)/FB Inputs/F{1..9 step 2} X-Field <-> Data Pointer/HallSensorFieldsXYZ[{75..87 step 3}]  (5 links)
//     Term 23 (APS4322-7000)/Term 24 (APS4322-5000)/FB Inputs/F{1..9 step 2} Y-Field <-> Data Pointer/HallSensorFieldsXYZ[{76..88 step 3}]  (5 links)
//     Term 23 (APS4322-7000)/Term 24 (APS4322-5000)/FB Inputs/F{1..9 step 2} Z-Field <-> Data Pointer/HallSensorFieldsXYZ[{77..89 step 3}]  (5 links)
//     Term 23 (APS4322-7000)/Term 24 (APS4322-5000)/FB Inputs/G{0..8 step 2} X-Field <-> Data Pointer/HallSensorFieldsXYZ[{90..102 step 3}]  (5 links)
//     Term 23 (APS4322-7000)/Term 24 (APS4322-5000)/FB Inputs/G{0..8 step 2} Y-Field <-> Data Pointer/HallSensorFieldsXYZ[{91..103 step 3}]  (5 links)
//     Term 23 (APS4322-7000)/Term 24 (APS4322-5000)/FB Inputs/G{0..8 step 2} Z-Field <-> Data Pointer/HallSensorFieldsXYZ[{92..104 step 3}]  (5 links)
//     Term 23 (APS4322-7000)/Term 24 (APS4322-5000)/FB Inputs/H{1..9 step 2} X-Field <-> Data Pointer/HallSensorFieldsXYZ[{105..117 step 3}]  (5 links)
//     Term 23 (APS4322-7000)/Term 24 (APS4322-5000)/FB Inputs/H{1..9 step 2} Y-Field <-> Data Pointer/HallSensorFieldsXYZ[{106..118 step 3}]  (5 links)
//     Term 23 (APS4322-7000)/Term 24 (APS4322-5000)/FB Inputs/H{1..9 step 2} Z-Field <-> Data Pointer/HallSensorFieldsXYZ[{107..119 step 3}]  (5 links)
//     Term 23 (APS4322-7000)/Term 24 (APS4322-5000)/FB Inputs/I{0..8 step 2} X-Field <-> Data Pointer/HallSensorFieldsXYZ[{120..132 step 3}]  (5 links)
//     Term 23 (APS4322-7000)/Term 24 (APS4322-5000)/FB Inputs/I{0..8 step 2} Y-Field <-> Data Pointer/HallSensorFieldsXYZ[{121..133 step 3}]  (5 links)
//     Term 23 (APS4322-7000)/Term 24 (APS4322-5000)/FB Inputs/I{0..8 step 2} Z-Field <-> Data Pointer/HallSensorFieldsXYZ[{122..134 step 3}]  (5 links)
//     Term 23 (APS4322-7000)/Term 24 (APS4322-5000)/FB Inputs/J{1..9 step 2} X-Field <-> Data Pointer/HallSensorFieldsXYZ[{135..147 step 3}]  (5 links)
//     Term 23 (APS4322-7000)/Term 24 (APS4322-5000)/FB Inputs/J{1..9 step 2} Y-Field <-> Data Pointer/HallSensorFieldsXYZ[{136..148 step 3}]  (5 links)
//     Term 23 (APS4322-7000)/Term 24 (APS4322-5000)/FB Inputs/J{1..9 step 2} Z-Field <-> Data Pointer/HallSensorFieldsXYZ[{137..149 step 3}]  (5 links)
//     Term 23 (APS4322-7000)/Term 24 (APS4322-5000)/FB Inputs/Status <-> Data Pointer/FeedbackStatus
//   XPlanar MC Project/Axes/0000kyte <-> TcCOM Objects/XPlanar/0000kyte
//     IoToMc/STD <-> OutputsToNC3/HWToNC3
//     McToIo/STD <-> InputsFromNC3/NC3ToHW
//   XPlanar MC Project/Axes/0000kytm <-> TcCOM Objects/XPlanar/0000kytm
//     IoToMc/STD <-> OutputsToNC3/HWToNC3
//     McToIo/STD <-> InputsFromNC3/NC3ToHW
//   XPlanar MC Project/Axes/0000kytn <-> TcCOM Objects/XPlanar/0000kytn
//     IoToMc/STD <-> OutputsToNC3/HWToNC3
//     McToIo/STD <-> InputsFromNC3/NC3ToHW
//   XPlanar MC Project/Axes/0000kyto <-> TcCOM Objects/XPlanar/0000kyto
//     IoToMc/STD <-> OutputsToNC3/HWToNC3
//     McToIo/STD <-> InputsFromNC3/NC3ToHW
//   SK12_StarterkitApplicationPLC_V3/SK12_StarterkitApplicationPLC_V3 Instance <-> Device 6 (USB)/Box 1 (CX2100 Power Supply)
//     PlcTask Inputs/MAIN.bCxButtonRingDown <-> DIS Inputs/Status/Down
//     PlcTask Inputs/MAIN.bCxButtonRingEnter <-> DIS Inputs/Status/Enter
//     PlcTask Inputs/MAIN.bCxButtonRingLeft <-> DIS Inputs/Status/Left
//     PlcTask Inputs/MAIN.bCxButtonRingRight <-> DIS Inputs/Status/Right
//     PlcTask Inputs/MAIN.bCxButtonRingToggle <-> DIS Inputs/Status/TxPDO Toggle
//     PlcTask Inputs/MAIN.bCxButtonRingUp <-> DIS Inputs/Status/Up
//   SK12_StarterkitApplicationPLC_V3/SK12_StarterkitApplicationPLC_V3 Instance <-> XPlanar MC Project/Axes/0000kyte
//     PlcTask Inputs/MAIN.fbXMotionUnit.fbXPlanarMover[1].stMoverRef.MCTOPLC/ACT <-> McToPlc/ACT
//     PlcTask Inputs/MAIN.fbXMotionUnit.fbXPlanarMover[1].stMoverRef.MCTOPLC/COORDMODE <-> McToPlc/COORDMODE
//     PlcTask Inputs/MAIN.fbXMotionUnit.fbXPlanarMover[1].stMoverRef.MCTOPLC/SET <-> McToPlc/SET
//     PlcTask Inputs/MAIN.fbXMotionUnit.fbXPlanarMover[1].stMoverRef.MCTOPLC/SETONTRACK <-> McToPlc/SETONTRACK
//     PlcTask Inputs/MAIN.fbXMotionUnit.fbXPlanarMover[1].stMoverRef.MCTOPLC/STD <-> McToPlc/STD
//     PlcTask Outputs/MAIN.fbXMotionUnit.fbXPlanarMover[1].stMoverRef.PLCTOMC/STD <-> PlcToMc/STD
//   SK12_StarterkitApplicationPLC_V3/SK12_StarterkitApplicationPLC_V3 Instance <-> XPlanar MC Project/Axes/0000kytm
//     PlcTask Inputs/MAIN.fbXMotionUnit.fbXPlanarMover[3].stMoverRef.MCTOPLC/ACT <-> McToPlc/ACT
//     PlcTask Inputs/MAIN.fbXMotionUnit.fbXPlanarMover[3].stMoverRef.MCTOPLC/COORDMODE <-> McToPlc/COORDMODE
//     PlcTask Inputs/MAIN.fbXMotionUnit.fbXPlanarMover[3].stMoverRef.MCTOPLC/SET <-> McToPlc/SET
//     PlcTask Inputs/MAIN.fbXMotionUnit.fbXPlanarMover[3].stMoverRef.MCTOPLC/SETONTRACK <-> McToPlc/SETONTRACK
//     PlcTask Inputs/MAIN.fbXMotionUnit.fbXPlanarMover[3].stMoverRef.MCTOPLC/STD <-> McToPlc/STD
//     PlcTask Outputs/MAIN.fbXMotionUnit.fbXPlanarMover[3].stMoverRef.PLCTOMC/STD <-> PlcToMc/STD
//   SK12_StarterkitApplicationPLC_V3/SK12_StarterkitApplicationPLC_V3 Instance <-> XPlanar MC Project/Axes/0000kytn
//     PlcTask Inputs/MAIN.fbXMotionUnit.fbXPlanarMover[4].stMoverRef.MCTOPLC/ACT <-> McToPlc/ACT
//     PlcTask Inputs/MAIN.fbXMotionUnit.fbXPlanarMover[4].stMoverRef.MCTOPLC/COORDMODE <-> McToPlc/COORDMODE
//     PlcTask Inputs/MAIN.fbXMotionUnit.fbXPlanarMover[4].stMoverRef.MCTOPLC/SET <-> McToPlc/SET
//     PlcTask Inputs/MAIN.fbXMotionUnit.fbXPlanarMover[4].stMoverRef.MCTOPLC/SETONTRACK <-> McToPlc/SETONTRACK
//     PlcTask Inputs/MAIN.fbXMotionUnit.fbXPlanarMover[4].stMoverRef.MCTOPLC/STD <-> McToPlc/STD
//     PlcTask Outputs/MAIN.fbXMotionUnit.fbXPlanarMover[4].stMoverRef.PLCTOMC/STD <-> PlcToMc/STD
//   SK12_StarterkitApplicationPLC_V3/SK12_StarterkitApplicationPLC_V3 Instance <-> XPlanar MC Project/Axes/0000kyto
//     PlcTask Inputs/MAIN.fbXMotionUnit.fbXPlanarMover[2].stMoverRef.MCTOPLC/ACT <-> McToPlc/ACT
//     PlcTask Inputs/MAIN.fbXMotionUnit.fbXPlanarMover[2].stMoverRef.MCTOPLC/COORDMODE <-> McToPlc/COORDMODE
//     PlcTask Inputs/MAIN.fbXMotionUnit.fbXPlanarMover[2].stMoverRef.MCTOPLC/SET <-> McToPlc/SET
//     PlcTask Inputs/MAIN.fbXMotionUnit.fbXPlanarMover[2].stMoverRef.MCTOPLC/SETONTRACK <-> McToPlc/SETONTRACK
//     PlcTask Inputs/MAIN.fbXMotionUnit.fbXPlanarMover[2].stMoverRef.MCTOPLC/STD <-> McToPlc/STD
//     PlcTask Outputs/MAIN.fbXMotionUnit.fbXPlanarMover[2].stMoverRef.PLCTOMC/STD <-> PlcToMc/STD
//   SK12_StarterkitApplicationPLC_V3/SK12_StarterkitApplicationPLC_V3 Instance <-> XPlanar MC Project/Groups/Environment
//     PlcTask Inputs/MAIN.fbXMotionUnit.fbXPlanarSystem.environment.MCTOPLC_STD <-> McToPlc/STD
//   SK12_StarterkitApplicationPLC_V3/SK12_StarterkitApplicationPLC_V3 Instance <-> XPlanar MC Project/Groups/Track1
//     PlcTask Inputs/MAIN.fbXMotionUnit.fbTrackSegment01.fbTrackStandard.stTrackRef.MCTOPLC_STD <-> McToPlc/STD
//   SK12_StarterkitApplicationPLC_V3/SK12_StarterkitApplicationPLC_V3 Instance <-> XPlanar MC Project/Groups/Track2
//     PlcTask Inputs/MAIN.fbXMotionUnit.fbTrackSegment02.fbTrackStandard.stTrackRef.MCTOPLC_STD <-> McToPlc/STD
//   SK12_StarterkitApplicationPLC_V3/SK12_StarterkitApplicationPLC_V3 Instance <-> XPlanar MC Project/Groups/Track3
//     PlcTask Inputs/MAIN.fbXMotionUnit.fbTrackSegment03.fbTrackStandard.stTrackRef.MCTOPLC_STD <-> McToPlc/STD
//   SK12_StarterkitApplicationPLC_V3/SK12_StarterkitApplicationPLC_V3 Instance <-> XPlanar MC Project/Groups/XPlanar
//     PlcTask Inputs/MAIN.fbXMotionUnit.fbXPlanarSystem.group.MCTOPLC_STD <-> McToPlc/STD

CONFIGURATION SK12_StarterkitApplicationPLC_V3
    RESOURCE PLC ON TwinCAT3
        TASK PlcTask(INTERVAL := T#10ms, PRIORITY := 16);
        PROGRAM MAIN WITH PlcTask : MAIN;
    END_RESOURCE
END_CONFIGURATION

// ---- 1_Industry/DUTs/E_XMotion_Command.TcDUT
{attribute 'qualified_only'}
{attribute 'strict'}
TYPE E_XMotion_Command :
(
	NoCommand		:= 0,
	Abort			:= 1,
	Reset			:= 2,
	Prepare			:= 3,
	Start			:= 4,
	HoldOnError		:= 5,
	UserCommand		:= 6
	
) DINT;
END_TYPE

// ---- 1_Industry/DUTs/E_XMotion_Status.TcDUT
{attribute 'qualified_only'}
{attribute 'strict'}
TYPE E_XMotion_Status :
(
	StartUp 	:= 0,
	Aborting 	:= 1,
	Aborted 	:= 2,	
	Resetting   := 3,
	Stopped  	:= 4,
	Preparing   := 5,
	Prepared    := 6,
	Execute 	:= 7,
	HoldOnError := 8
	
) DINT;
END_TYPE

// ---- 1_Industry/DUTs/ST_VisControl.TcDUT
TYPE ST_VisControl :
STRUCT
	
	stControlPad	: ST_Vis_ControlPadControl;
	stOperatorPad	: ST_Vis_OperationalControl;


END_STRUCT
END_TYPE

// ---- 1_Industry/DUTs/ST_Vis_ControlPadControl.TcDUT
TYPE ST_Vis_ControlPadControl :
STRUCT
	
	bVisInvisibleButton	: BOOL;	
	bVisInvisible		: BOOL;	
	nFramePositionX		: INT;
	nFramePositionY		: INT;
	nButtonPositionX	: INT;
	nButtonPositionY	: INT;
	
	bButtonState_Abort			: BOOL;
	bButtonState_Reset			: BOOL;
	bButtonState_Prepare		: BOOL;	
	bButtonState_Start			: BOOL;
	
	bStateSignalAbortBlue		: BOOL;
	bStateSignalAbortYellow		: BOOL;
	bStateSignalAbortGreen		: BOOL;
	
	bStateSignalResetYellow		: BOOL;
	bStateSignalResetGreen		: BOOL;

	bStateSignalPrepareYellow	: BOOL;
	bStateSignalPrepareGreen	: BOOL;

	bStateSignalExecuteYellow	: BOOL;
	bStateSignalExecuteGreen	: BOOL;	

	bAbortSequenceStateInvisible	: BOOL;
	bResetSequenceStateInvisible	: BOOL;
	bPrepareSequenceStateInvisible	: BOOL;
	bStartSequenceStateInvisible	: BOOL;
	
	iAbortSequenceState			: INT;
	iResetSequenceState			: INT;
	iPrepareSequenceState		: INT;
	iStartSequenceState			: INT;	
	
	
END_STRUCT
END_TYPE

// ---- 1_Industry/DUTs/ST_Vis_OperationalControl.TcDUT
TYPE ST_Vis_OperationalControl :
STRUCT
	bVisInvisibleButton	: BOOL;	
	bVisInvisible		: BOOL;
	nFramePositionX		: REAL;
	nFramePositionY		: REAL;
	nButtonPositionX	: INT;
	nButtonPositionY	: INT;	
	
	bStartButtunState	: BOOL;
	bStopButtonState	: BOOL;
	bQuitButtonState	: BOOL;
	bEStopButtonState	: BOOL;
	
	bStartButtonLamp	: BOOL;
	bStopButtonLamp		: BOOL;
	bQuitButtonLamp		: BOOL;
	bEStopButtonLamp	: BOOL;
	
	bMessageColorGreen	: BOOL;
	bMessageColorRed	: BOOL;
	
	sMessage			: STRING;
	
	
END_STRUCT
END_TYPE

// ---- 1_Industry/DUTs/ST_XMotionStatemachineStates.TcDUT
TYPE ST_XMotionStatemachineStates :
STRUCT
	nAbortState		: INT;
	nResetState		: INT;
	nPrepareState	: INT;
	nStartState		: INT;
END_STRUCT
END_TYPE

// ---- 1_Industry/DUTs/ST_XTags.TcDUT
TYPE ST_XTags :
STRUCT
	

	Command		: E_XMotion_Command;
	Status		: E_XMotion_Status;
	States		: ST_XMotionStatemachineStates;
	
END_STRUCT
END_TYPE

// ---- 2_Application/Machine/DUTs/ST_MessageBoxText.TcDUT
TYPE ST_MessageBoxText :
STRUCT
	
	sText	: STRING;
	nColor	: DWORD;	

END_STRUCT
END_TYPE

// ---- 2_Application/Machine/DUTs/ST_VisuMessage.TcDUT
TYPE ST_VisuMessage :
STRUCT

	bVisible_Box1_A		: BOOL;
	bVisible_Box1_B		: BOOL;	
	
	sMessage_L1_Box1	: ST_MessageBoxText;
	sMessage_L2_Box1	: ST_MessageBoxText;
	
	bAcknowledge		: BOOL;
	
END_STRUCT
END_TYPE

// ---- 2_Application/Machine/DUTs/ST_MachineState.TcDUT
TYPE ST_MachineState :
STRUCT

	bStartup	 : BOOL;		
	bStartupDone : BOOL;
	bAborting 	 : BOOL;
	bResetting	 : BOOL;
	bStarting	 : BOOL;
	bRunning	 : BOOL;

END_STRUCT
END_TYPE

// ---- 2_Application/Machine/DUTs/ST_MoverDistance.TcDUT
TYPE ST_MoverDistance :
STRUCT
	nPositionIndex	: UDINT;
	fDistance		: LREAL;
END_STRUCT
END_TYPE

// ---- 2_Application/Machine/DUTs/ST_PositionXY.TcDUT
TYPE ST_PositionXY :
STRUCT
	x 		: LREAL;
	Y 		: LREAL;
	valid 	: BOOL;
END_STRUCT
END_TYPE

// ---- 2_Application/Mover/DUTs/ST_ProductData.TcDUT
TYPE ST_ProductData :
STRUCT
	
	nSerial				: UDINT;
	bInitRun			: BOOL;
	nDestinationProcess	: UINT;
	nPriority			: UINT;
	

END_STRUCT
END_TYPE

// ---- 2_Application/Station/DUTs/E_ProcessMode.TcDUT
{attribute 'qualified_only'}
{attribute 'strict'}
TYPE E_ProcessMode :
(
	None        := 0,
	InitRun	    := 1,
	Production	:= 2
	
);
END_TYPE

// ---- 2_Application/Station/DUTs/ST_StationPosition.TcDUT
TYPE ST_StationPosition :
STRUCT
	bInit				: BOOL;
	fPositionOnTrack	: LREAL;
	nTrackId			: UINT;
	fPosition_X			: LREAL;
	fPosition_Y			: LREAL;
END_STRUCT
END_TYPE

// ---- 2_Application/Station/DUTs/ST_StationReturn.TcDUT
TYPE ST_StationReturn :
STRUCT
	Done	: BOOL;
	stState	: INT;
END_STRUCT
END_TYPE

// ---- 2_Application/Station/DUTs/ST_VisStationData.TcDUT
TYPE ST_VisStationData :

STRUCT
	
	bInit		: BOOL;
	fPosition_X	: LREAL;
	fPosition_Y : LREAL;

END_STRUCT

END_TYPE

// ---- 1_Industry/GlobalVariables.TcGVL


VAR_GLOBAL
	
	XTags			: ST_XTags;		

	stVisControl	: ST_VisControl;
	

END_VAR

// ---- 2_Application/GVL_Application.TcGVL
VAR_GLOBAL CONSTANT
	
	gc_nMaxNumberMovers			: UDINT := 4;	
	gc_nMoverCountConfigured 	: UDINT := gc_nMaxNumberMovers;
	
	gc_MaxNumberTiles			: UDINT := 24;

	gc_NumberTracks				: UDINT := 3;		// Number of tracks controlled by the application
	gc_NumberStations			: UINT  := 5;		// Number of stations controlled by the application
	gc_MaxNumberTrackPoints		: INT   := 20;		// max number of track points for each track 
END_VAR

VAR_GLOBAL
	g_nMoverCount				: UDINT := 4;
	g_nMoverCountPresent		: UDINT := g_nMoverCount;
	
	ipTrack						: ARRAY [1..gc_NumberTracks] OF I_Track;
	ipStation					: ARRAY [1..gc_NumberStations] OF I_Station;
	ipMoverApplication			: ARRAY [1..gc_nMaxNumberMovers] OF I_MoverApplication;
	ipMotionSystemApplication	: I_MotionSystemApplication;

	g_VisStationData			: ARRAY[1..gc_NumberStations] OF ST_VisStationData;
	
	
	sTextTemp					: STRING;
	ipVisuMessage				: I_VisuMessage;				
	g_VisuMessage				: ST_VisuMessage;
END_VAR

// ---- 2_Application/Machine/I_MotionSystemApplication.TcIO
INTERFACE I_MotionSystemApplication

METHOD Aborting : BOOL
VAR_INPUT
END_VAR
END_METHOD

METHOD Cycle : BOOL
VAR_INPUT
END_VAR
END_METHOD

METHOD Execute : UDINT
VAR_INPUT
END_VAR
END_METHOD

PROPERTY PUBLIC P_AbortingSequence : DINT
GET
END_GET
END_PROPERTY

PROPERTY P_Alarm : ST_VisuMessage
GET
END_GET
END_PROPERTY

PROPERTY PUBLIC P_ExecutingSequence : DINT
GET
END_GET
END_PROPERTY

PROPERTY P_MoverError : BOOL
GET
END_GET
SET
END_SET
END_PROPERTY

PROPERTY PUBLIC P_ResettingSequence : DINT
GET
END_GET
END_PROPERTY

PROPERTY PUBLIC P_StartingSequence : DINT
GET
END_GET
END_PROPERTY

PROPERTY PUBLIC P_StartupSequence : DINT
GET
END_GET
END_PROPERTY

METHOD Prepare : BOOL
VAR_INPUT
END_VAR
END_METHOD

METHOD Reset : BOOL
VAR_INPUT
END_VAR
END_METHOD

METHOD Resetting : BOOL
END_METHOD

METHOD Startup : BOOL
VAR_INPUT
END_VAR
END_METHOD

PROPERTY std : I_MotionSystem
GET
END_GET
SET
END_SET
END_PROPERTY

END_INTERFACE

// ---- 2_Application/Mover/I_MoverApplication.TcIO
INTERFACE I_MoverApplication

METHOD Cycle
END_METHOD

PROPERTY P_MoverIndex : INT
GET
END_GET
SET
END_SET
END_PROPERTY

PROPERTY P_ProductData : Reference to ST_ProductData
GET
END_GET
SET
END_SET
END_PROPERTY

PROPERTY P_TrackId : UDINT
GET
END_GET
SET
END_SET
END_PROPERTY

PROPERTY std : I_XPlanarMoverStandard
GET
END_GET
SET
END_SET
END_PROPERTY

END_INTERFACE

// ---- 2_Application/Station/Base/I_Station.TcIO
INTERFACE I_Station

METHOD Clear : BOOL
VAR_INPUT
END_VAR
END_METHOD

METHOD Cycle : BOOL
VAR_INPUT
END_VAR
END_METHOD

METHOD Init : BOOL
END_METHOD

PROPERTY P_bInitDone : BOOL
GET
END_GET
END_PROPERTY

PROPERTY P_eProcessMode : E_ProcessMode
GET
END_GET
SET
END_SET
END_PROPERTY

PROPERTY P_List_Station : I_List
GET
END_GET
END_PROPERTY

PROPERTY P_List_Switch_Input_A : I_List
GET
END_GET
END_PROPERTY

PROPERTY P_List_Switch_Input_B : I_List
GET
END_GET
END_PROPERTY

PROPERTY P_List_Switch_Input_C : I_List
GET
END_GET
END_PROPERTY

PROPERTY P_nErrorCode : UDINT
GET
END_GET
END_PROPERTY

PROPERTY P_Position : ST_StationPosition
GET
END_GET
END_PROPERTY

PROPERTY P_ProcessClearance : DINT
GET
END_GET
END_PROPERTY

PROPERTY P_ProcessRequest : DINT
GET
END_GET
SET
END_SET
END_PROPERTY

PROPERTY P_ProcessState : DINT
GET
END_GET
END_PROPERTY

METHOD Process : BOOL
END_METHOD

END_INTERFACE

// ---- 2_Application/Tracks/Base/I_Track.TcIO
INTERFACE I_Track

METHOD Clear : BOOL
END_METHOD

METHOD Cycle : BOOL
END_METHOD

METHOD Initialize : BOOL
VAR_INPUT
	nTrackIndex : UDINT;
END_VAR
END_METHOD

PROPERTY P_Error : BOOL
GET
END_GET
END_PROPERTY

PROPERTY P_ErrorInfo : STRING
GET
END_GET
END_PROPERTY

PROPERTY P_TrackLength : LREAL
GET
END_GET
END_PROPERTY

PROPERTY std : I_TrackStandard
GET
END_GET
END_PROPERTY

END_INTERFACE

// ---- VISU/Logic/I_VisuMessage.TcIO
INTERFACE I_VisuMessage

METHOD CheckAknowledge : BOOL
VAR_INPUT
END_VAR
END_METHOD

METHOD ClearAlarmMessage : BOOL
VAR_INPUT
END_VAR
END_METHOD

METHOD ClearAllMessages : BOOL
VAR_INPUT
END_VAR
END_METHOD

METHOD ClearInfoMessage : BOOL
VAR_INPUT
END_VAR
END_METHOD

METHOD SetAlarmMessage : BOOL
VAR_INPUT
	sMessage	: STRING;
END_VAR
END_METHOD

METHOD SetErrorMessage : BOOL
VAR_INPUT
	sMessage	: STRING;
	sSequence	: STRING;
	nState		: DINT;
	nErrorCode	: DWORD;
END_VAR
END_METHOD

METHOD SetInfoMessage : BOOL
VAR_INPUT
	sMessage	: STRING;
	sSequence	: STRING;
	nState		: DINT;
END_VAR
END_METHOD

METHOD StateUpdate : BOOL
VAR_INPUT
	nState		: DINT;
	sSequence	: STRING;
END_VAR
END_METHOD

END_INTERFACE

// ---- MAIN.TcPOU
{attribute 'TcCallAfterOutputUpdate'}
PROGRAM MAIN

VAR
	fbXMotionUnit					: FB_MachineModule;
	fbOperationalControl			: FB_OperationalControl;
	fbVisStarterKitStateMachine		: FB_VisStarterKitStateMachine;	
	
	stVisAlarm						: ST_VisuMessage;	

	nTestCNT	: UINT;
END_VAR
	

VAR
    bCxButtonRingUp 		AT %I* 	: BOOL;
    bCxButtonRingDown		AT %I*	: BOOL;
    bCxButtonRingLeft 		AT %I*  : BOOL;
    bCxButtonRingRight 		AT %I*  : BOOL;
    bCxButtonRingEnter 		AT %I* 	: BOOL;
    bCxButtonRingToggle 	AT %I*  : BOOL;
END_VAR



Cycle();


nTestCNT := nTestCNT +1;

METHOD Cycle : BOOL
VAR_INPUT
END_VAR


VAR
	bExternalMachineStop 	: BOOL;	
	bHelp01					: BOOL;
	bHelp02					: BOOL;	
	bHelp03					: BOOL;
	bHelp04					: BOOL;	
	sHelp01					: STRING;
	nHelp01					: INT;	
	bResetOC				: BOOL;
	idx						: UDINT;
	stPosition				: ST_StationPosition;
END_VAR


	// Keeping the motion system alive
	fbXMotionUnit.Cycle(); 	
	stVisAlarm := fbXMotionUnit.P_Alarm;								   

	
	// Exchanging XTags and Commands 
	XTags.Status := fbXMotionUnit.P_XMotionStatus;			// Getting current status of XMotionUnit for e.g. HMI display	
	XTags.States := fbXMotionUnit.P_XSequenceStates; 		// Writing current states information into XTags
	
	fbXMotionUnit.P_XCommand 	 := XTags.Command;	    								// Writing command from superior unit e.g. HMI
	fbXMotionUnit.P_ExternelStop := bExternalMachineStop;								// External exception e.g. signal from E-Stop	
	fbXMotionUnit.P_ErrorQuit    := fbVisStarterKitStateMachine.P_OCQuitButtonState;	// Error-Quit from external button
	
	
	// Operational Control 		
	IF XTags.Status = E_XMotion_Status.Aborting 
	OR XTags.Status = E_XMotion_Status.Aborted
	THEN
		bResetOC := TRUE;
	ELSE
		bResetOC := FALSE;
	END_IF
	fbOperationalControl.P_ProcessFeedback := fbXMotionUnit.P_ProcessFeedback;
	
	fbOperationalControl(	   bStartCommand := fbVisStarterKitStateMachine.P_OCStartButtonState OR bCxButtonRingUp, 
								bStopCommand := fbVisStarterKitStateMachine.P_OCStopButtonState OR bCxButtonRingDown, 
								bQuitCommand := fbVisStarterKitStateMachine.P_OCQuitButtonState OR bCxButtonRingEnter,
						   bExceptionCommand := fbVisStarterKitStateMachine.P_OCEStopButtonState,
							   bResetCommand := bResetOC,
								  bStartLamp => bHelp01,
								   bStopLamp => bHelp02,
								   bQuitLamp => bHelp03,
								  bEStopLamp => bHelp04,
									bStopped => ,
								   bStarting => , 
									bRunning => , 
									 sResult => sHelp01,
									 nResult => nHelp01,
									   XTags := XTags );
		
	
								fbVisStarterKitStateMachine.P_OCStartLampState 		:= bHelp01;
								fbVisStarterKitStateMachine.P_OCStopLampState  		:= bHelp02;
								fbVisStarterKitStateMachine.P_OCQuitLampState  		:= bHelp03;
								fbVisStarterKitStateMachine.P_OCEStopLampState  	:= bHelp04;
								fbVisStarterKitStateMachine.P_OCResultTextDisplay 	:= sHelp01;
								fbVisStarterKitStateMachine.P_OCResult 				:= nHelp01;							  
	
								
	// Visu Statemachine									  
	fbVisStarterKitStateMachine( iq_stVisControl := stVisControl,
										iq_XTags := XTags );
	
	
	// Collecting station data for visulization
	FOR idx:=1 TO gc_NumberStations DO
		IF ipStation[idx] <> 0 THEN
			stPosition := ipStation[idx].P_Position;
			g_VisStationData[idx].bInit       := stPosition.bInit;
			g_VisStationData[idx].fPosition_X := stPosition.fPosition_X;
			g_VisStationData[idx].fPosition_Y := stPosition.fPosition_Y;
		END_IF
	END_FOR
END_METHOD

END_PROGRAM

// ---- 1_Industry/FB_MachineModule.TcPOU
FUNCTION_BLOCK FB_MachineModule 

VAR
//===== Aplication Layer =================================

	fbMotionSystem			: FB_MotionSystem;
	fbXPlanarSystem			: FB_XPlanarSystem;
	
	fbMover					: ARRAY [1..gc_nMaxNumberMovers] OF FB_ApplicationMover;
	fbXPlanarMover			: ARRAY [1..gc_nMaxNumberMovers] OF FB_XPlanarMoverStandard; 
	
	fbVisuMessage			: FB_VisuMessage;
	
	// Instances of Track-FBs
	fbTrackSegment01		: FB_TrackSegment_1;
	fbTrackSegment02		: FB_TrackSegment_2;
	fbTrackSegment03		: FB_TrackSegment_3;
	   
	// Instances of Station-FBs
	fbStation_01_Process 	: FB_Station_01_Process;
	fbStation_02_Process 	: FB_Station_02_Process;
	fbStation_03_Process	: FB_Station_03_Process;
	fbStation_04_Switch		: FB_Station_04_SW_Separate;
	fbStation_05_Switch		: FB_Station_05_SW_Merge;
	
//===== Base Module =======================================

	eXCommand					: E_XMotion_Command;
	eXStatus					: E_XMotion_Status;
	eLastXState					: E_XMotion_Status;	

	fbStateManager				: FB_SK_StateManager;
	eControlCommand				: E_XMotion_Command;
	stSequenceStates 			: ST_XMotionStatemachineStates;
	stAlarm						: ST_VisuMessage;
	
	nStateCommandCheck			: INT;
	bMachineExceptionPending	: BOOL;
	
	bUnitModeManagerExecute		: BOOL;
	bUnitModeManagerDone		: BOOL;
	bUnitModeManagerError		: BOOL;
		
	nStateSequence				: INT;
	nStateExecute				: INT;
	bInterfaceAssignmentDone	: BOOL;
	bDone						: BOOL;
	
	nProcessFeedback			: UDINT;
	bErrorQuit					: BOOL;
	
	nForCounter					: UDINT;

	fbVisuDignostics 			: FB_XPlanarVisuDiag;
	bVisuDiagInit				: BOOL;
	bVisuDiagInitMover 			: BOOL;
	bVisuDiagInitTrack 			: BOOL;

	
	// ...just for testing 
	nTestCounter_Cycle				: UINT;
	nTestCounter_Aborted			: UINT;
	nTestCounter_Aborting			: UINT;
	nTestCounter_Execute			: UINT;
	nTestCounter_Preparing			: UINT;
	nTestCounter_Prepared			: UINT;
	nTestCounter_Resetting 			: UINT;
	nTestCounter_StartUp			: UINT;
	nTestCounter_StateComplete 		: UINT;
	nTestCounter_Stopped			: UINT;
	nTestCounter_CommandReceive		: UINT;	
	
END_VAR

{attribute 'object_name' := 'Aborted'}
METHOD PRIVATE Aborted



	nTestCounter_Aborted := nTestCounter_Aborted + 1;
	
	(*
		Aborted:
		- all movers deactivated
		- No errors pending
	*)
END_METHOD

{attribute 'object_name' := 'Aborting'}
METHOD PRIVATE Aborting
CASE nStateSequence OF
	0: 		
		IF ipMotionSystemApplication <> 0 THEN
			nStateSequence := 10;
		END_IF


	10:	
		IF ipMotionSystemApplication.Aborting() THEN
			nStateSequence := 100;
		END_IF

	100:
		StateComplete();
END_CASE
END_METHOD

METHOD PRIVATE CommandReceive 
VAR_INPUT
END_VAR


	nTestCounter_CommandReceive := nTestCounter_CommandReceive + 1;


	
	// Checking Statecommands and reacting to received Control-Commands
	CASE nStateCommandCheck OF
	
	
	0:  // Check
		IF NOT bMachineExceptionPending THEN
			nStateCommandCheck:= 10;   	// No error
		ELSE
			nStateCommandCheck:= 20;	// Error pending
		END_IF
	
		
	10:	// No Machine-Error 
		
		CASE eXCommand OF 		// XTags.eCommand received from superior system e.g. Machine-HMI

		E_XMotion_Command.NoCommand:
				eControlCommand := E_XMotion_Command.NoCommand;
		
		E_XMotion_Command.Abort:
				eControlCommand := E_XMotion_Command.Abort;
		
		E_XMotion_Command.Reset: 
				IF eXStatus = E_XMotion_Status.Aborted THEN
					eControlCommand := E_XMotion_Command.Reset;
				END_IF		
		
		E_XMotion_Command.Prepare:
				IF eXStatus = E_XMotion_Status.Stopped THEN
					eControlCommand := E_XMotion_Command.Prepare;
				END_IF
	
		E_XMotion_Command.Start:	
				IF eXStatus = E_XMotion_Status.Prepared THEN
					eControlCommand := E_XMotion_Command.Start;
				END_IF		
			
		E_XMotion_Command.HoldOnError:
				eControlCommand := E_XMotion_Command.HoldOnError;

				
		E_XMotion_Command.UserCommand:
				;
		
		// Rückmeldung wenn/warum ein Command nicht ausgeführt wurde		
							
		END_CASE
				
		nStateCommandCheck := 0;	
	
		
	20:  // Machine-Error reaction
		   eControlCommand := E_XMotion_Command.Abort;
		nStateCommandCheck := nStateCommandCheck + 1;	
		
	21: IF XTags.Status = E_XMotion_Status.Aborted THEN
			nStateCommandCheck := nStateCommandCheck + 1;
		END_IF		
			
	22:	IF NOT bMachineExceptionPending THEN
			nStateCommandCheck := 10;
		END_IF
		
		
	END_CASE
END_METHOD

METHOD PUBLIC Cycle
VAR
	nForCounter : UDINT;	
END_VAR


VAR_INST
	nTestCounter	 : UINT;
END_VAR
	nTestCounter := nTestCounter +1;


	fbMotionSystem.std := THIS^.fbXPlanarSystem;


	// Calling the state management of the main state-machine	
	StateManagement();


	// Keeping all cyclic activities alive and up-to-date
	IF ipMotionSystemApplication <> 0 THEN
		ipMotionSystemApplication.Cycle();
		stAlarm := ipMotionSystemApplication.P_Alarm;
	END_IF

	
	FOR nForCounter := 1 TO g_nMoverCount DO
		IF ipMoverApplication[nForCounter] <> 0 THEN
			ipMotionSystemApplication.std.SetMoverStandard(nForCounter, ipMoverApplication[nForCounter].std);
			ipMoverApplication[nForCounter].std.P_Id := UDINT_TO_UINT(nForCounter);
			ipMoverApplication[nforcounter].Cycle();		
		END_IF
	END_FOR	
	
	FOR nForCounter := 1 TO gc_NumberTracks DO
		IF ipTrack[nForCounter] <> 0 THEN
			ipMotionSystemApplication.std.SetTrackStandard(nForCounter, ipTrack[nForCounter].std);
			ipTrack[nForCounter].Cycle();
		END_IF
	END_FOR

	FOR nForCounter:=1 TO gc_NumberStations DO 
		IF ipStation[nForCounter] <> 0 THEN 
			ipStation[nForCounter].Cycle(); 
		END_IF
	END_FOR	
	
	
	// Logging/Diagnostics
	IF NOT bVisuDiagInit THEN
		
		IF NOT bVisuDiagInitMover THEN
			bVisuDiagInitMover := TRUE;
			FOR nForCounter := 1 TO g_nMoverCount DO 
				IF ipMoverApplication[nForCounter] <> 0 THEN
					fbVisuDignostics.SetStandardMover(ipMoverApplication[nForCounter].std, nForCounter);
				ELSE
					bVisuDiagInitMover := FALSE;
				END_IF
			END_FOR
		END_IF

		IF NOT bVisuDiagInitTrack THEN
			bVisuDiagInitTrack := TRUE;
			FOR nForCounter := 1 TO gc_NumberTracks DO 
				IF ipTrack[nForCounter] <> 0 THEN
					fbVisuDignostics.SetStandardTrack(ipTrack[nForCounter].std, nForCounter);
				ELSE
					bVisuDiagInitTrack := FALSE;
				END_IF
			END_FOR			
		END_IF
		
		bVisuDiagInit := bVisuDiagInitMover AND bVisuDiagInitTrack;
	END_IF
	
	

	fbVisuDignostics.Cycle();
	
	fbVisuMessage.Cycle(g_VisuMessage.bAcknowledge);
	g_VisuMessage := fbVisuMessage.P_VisuOut;
END_METHOD

{attribute 'object_name' := 'Execute'}
METHOD PRIVATE Execute


	
VAR_INST
	nForCounter : UDINT;	


END_VAR
	
	FOR nForCounter:=1 TO gc_NumberStations DO
		IF ipStation[nForCounter] <> 0 THEN
			ipStation[nForCounter].Process();
			
			IF ipStation[nForCounter].P_nErrorCode > 0 THEN
				nProcessFeedback := ipStation[nForCounter].P_nErrorCode;
			END_IF
		END_IF
	END_FOR	

	ipMotionSystemApplication.Execute();
	

	(*
	StateComplete();	// <- nothing will happen since there's no state defined after Execute,
						//    instead Execute can only be left by the Operator pressing the Abort-Button.
	*)
END_METHOD

METHOD HoldOnError : BOOL
VAR_INPUT
END_VAR



CASE nStateSequence OF
	0: 		
		IF ipMotionSystemApplication <> 0 THEN
			nStateSequence := 10;
		END_IF

	10:	
		IF nProcessFeedback = 0 THEN
			nStateSequence := 100;
		END_IF

	100:
		StateComplete();
END_CASE
END_METHOD

PROPERTY P_Alarm : ST_VisuMessage
GET
P_Alarm := stAlarm;
END_GET
END_PROPERTY

PROPERTY P_ErrorQuit : BOOL
SET
bErrorQuit := P_ErrorQuit;
END_SET
END_PROPERTY

PROPERTY P_ExternelStop : BOOL
GET
END_GET
SET
END_SET
END_PROPERTY

PROPERTY P_ProcessFeedback : UDINT
GET
P_ProcessFeedback := nProcessFeedback;
END_GET
END_PROPERTY

PROPERTY PUBLIC P_XCommand : E_XMotion_Command
SET
  eXCommand := P_XCommand;
END_SET
END_PROPERTY

PROPERTY PUBLIC P_XMotionStatus : E_XMotion_Status
GET
   P_XMotionStatus := eXStatus;
END_GET
END_PROPERTY

PROPERTY P_XSequenceStates : ST_XMotionStatemachineStates
GET
P_XSequenceStates := stSequenceStates;
END_GET
END_PROPERTY

METHOD PRIVATE Prepared
VAR_INPUT
END_VAR


	nTestCounter_Prepared := nTestCounter_Prepared +1;
	
	
	(*
		Prepared: 
		- all movers active (flying)
		- all movers in home position
	
	*)
END_METHOD

{attribute 'object_name' := 'Preparing'}
METHOD PRIVATE Preparing
CASE nStateSequence OF
	
	0: 		
		FOR nForCounter:=1 TO gc_NumberStations DO
			IF ipStation[nForCounter] <> 0 THEN
				ipStation[nForCounter].Process();				
				IF ipStation[nForCounter].P_nErrorCode > 0 THEN
					nProcessFeedback := ipStation[nForCounter].P_nErrorCode;
				END_IF
			END_IF
		END_FOR	
		

		IF ipMotionSystemApplication.Prepare() THEN
			nStateSequence := 100;
		END_IF

	100:
		StateComplete();
		
END_CASE
END_METHOD

{attribute 'object_name' := 'Resetting'}
METHOD PRIVATE Resetting

CASE nStateSequence OF
	
	0: 
		IF ipMotionSystemApplication.Resetting() THEN
			nStateSequence := 100;
		END_IF

		
	100:
		StateComplete();
		
END_CASE
END_METHOD

{attribute 'object_name' := 'StartUp'}
METHOD PRIVATE StartUp
VAR
	nForCounter : UDINT;
END_VAR
CASE nStateSequence OF

	0: 	// XPlanar- or XTS-System?
		ipVisuMessage := fbVisuMessage;
		fbMotionSystem.std := THIS^.fbXPlanarSystem;
		nStateSequence := 1;
		
	1:  // Mover assignment 
		FOR nForCounter := 1 TO g_nMoverCount DO
			fbMover[nForCounter].std := THIS^.fbXPlanarMover[nForCounter];
		END_FOR	
		nStateSequence := 2;
	
	2:	// Motion system to global motion system interface
		ipMotionSystemApplication := THIS^.fbMotionSystem;
		nStateSequence := 3;
			
	3:  // Movers to global mover interface
		FOR nForCounter := 1 TO g_nMoverCount DO
			ipMoverApplication[nForCounter] := THIS^.fbMover[nForCounter];
			THIS^.fbMover[nForCounter].P_MoverIndex := UDINT_TO_INT(nForCounter); 
		END_FOR	
		nStateSequence := 4;

	4:  // Assigning global Track-Interfaces
		ipTrack[1] := THIS^.fbTrackSegment01;
		ipTrack[2] := THIS^.fbTrackSegment02;
		ipTrack[3] := THIS^.fbTrackSegment03;	
		nStateSequence := 5;	
					
	5:  // Assigning global Station-Interfaces
		ipStation[1] := THIS^.fbStation_01_Process;
        ipStation[2] := THIS^.fbStation_02_Process;		
        ipStation[3] := THIS^.fbStation_03_Process;			
		ipStation[4] := THIS^.fbStation_04_Switch;
		ipStation[5] := THIS^.fbStation_05_Switch;	
	
		bInterfaceAssignmentDone := TRUE;
		nStateSequence := 10;
	
	
	10: // Calling Application-Startup-Procedure	
		IF ipMotionSystemApplication.Startup() THEN
			nStateSequence := 100;
		END_IF
	

	100: // Start-up done
		StateComplete();
END_CASE
END_METHOD

{attribute 'object_name' := 'StateComplete'}
METHOD PRIVATE StateComplete

	nTestCounter_StateComplete := nTestCounter_StateComplete + 1;

	nStateSequence := 0;
	
	//the actual state is completed
	fbStateManager.StateComplete();
END_METHOD

METHOD PRIVATE StateManagement : BOOL
VAR_INPUT
END_VAR
	// Checking for command received by superior unit e.g. HMI
	CommandReceive();
	
	
	// fbStateManager manages the state to be executed:
	fbStateManager.Cycle();	
	fbStateManager.XMotionCommand := eControlCommand;
	eXStatus := fbStateManager.Status;
						
	IF eXStatus <> eLastXState THEN
		nStateSequence := 0;
		eLastXState := eXStatus;
	END_IF

	
	// One of the methods is executing by the actual status
	CASE eXStatus OF
		E_XMotion_Status.StartUp:	        StartUp();
		E_XMotion_Status.Aborting:         Aborting();
		E_XMotion_Status.Aborted:           Aborted();
		E_XMotion_Status.Resetting:       Resetting();
		E_XMotion_Status.Stopped:           Stopped();
		E_XMotion_Status.Preparing:       Preparing();
		E_XMotion_Status.Prepared:         Prepared();
		E_XMotion_Status.Execute:	   		Execute();
		E_XMotion_Status.HoldOnError:	HoldOnError();
	END_CASE
	
	
	// Information to visulization etc.
	IF ipMotionSystemApplication <> 0 THEN 
		stSequenceStates.nAbortState   := DINT_TO_INT(ipMotionSystemApplication.P_AbortingSequence); 
		stSequenceStates.nResetState   := DINT_TO_INT(ipMotionSystemApplication.P_ResettingSequence);
		stSequenceStates.nPrepareState := DINT_TO_INT(ipMotionSystemApplication.P_StartingSequence);
		stSequenceStates.nStartState   := DINT_TO_INT(ipMotionSystemApplication.P_ExecutingSequence);
	END_IF
END_METHOD

{attribute 'object_name' := 'Stopped'}
METHOD PRIVATE Stopped

	nTestCounter_Stopped := nTestCounter_Stopped + 1;


	(*
	
		Stopped: 
		- Production finished
		- …
		
	*)
END_METHOD

END_FUNCTION_BLOCK

// ---- 2_Application/Machine/FB_MotionSystem.TcPOU
FUNCTION_BLOCK FB_MotionSystem IMPLEMENTS I_MotionSystemApplication

VAR
	
	ipMotionSystem			: I_MotionSystem;
	stMoverDetectionInfos   : ST_TcIoMoverDetectionInfos;
	
	// Sequences
	nStartupSequence 		: DINT;
	nAbortingSequence 		: DINT;
	nPrepareSequence 		: DINT;
	nResettingSequence 		: DINT;
	nExecutingSequence 		: DINT;	
	
	// Helper
	bDone 					: BOOL;
	idx						: UDINT;
	nForCounter 			: UDINT;	
	nErrorID				: UDINT;
	bMoverError				: BOOL;	

	
END_VAR

METHOD Aborting : BOOL
VAR_INST
	bWaitForRotatioFinished		: BOOL;
END_VAR

nErrorID := 0;

CASE nAbortingSequence OF 

	0: // Enter	
		bWaitForRotatioFinished := FALSE;
		FOR idx:=1 TO g_nMoverCount DO
			IF ipMoverApplication[idx].std.P_MoveC.Busy THEN
				bWaitForRotatioFinished := TRUE;	
			END_IF
		END_FOR
		
		IF NOT bWaitForRotatioFinished THEN
			nAbortingSequence := 10; 
		ELSE
			ipVisuMessage.SetInfoMessage('Waiting for rotation finished', 'Aborting', nAbortingSequence);	
		END_IF			
		
		
	10: // Sending "Halt" to all movers for immediate stop 
		IF ipMotionSystem.HaltSystem() THEN
			ipVisuMessage.SetInfoMessage('Sending HALT', 'Aborting', nAbortingSequence);
			nAbortingSequence := nAbortingSequence +1;
		END_IF
		
	11: IF ipMotionSystem.P_HaltSystem.Done THEN
			nAbortingSequence := nAbortingSequence +9;
		ELSIF ipMotionSystem.P_HaltSystem.Error THEN
			nAbortingSequence := nAbortingSequence +1;				
		END_IF
	
	12:	// Check error ID and react accordingly
		nErrorID := ipMotionSystem.P_HaltSystem.ErrorID;
		IF nErrorID = 33105 THEN
			nAbortingSequence := nAbortingSequence +8;
		ELSE
			ipVisuMessage.SetErrorMessage('HALT failed', 'Aborting', nAbortingSequence, nErrorID);
		END_IF
				

		
	20: // Reset Movers
		IF ipMotionSystem.ResetMovers() THEN
			ipVisuMessage.SetInfoMessage('RESET Movers', 'Aborting', nAbortingSequence);
			nAbortingSequence := nAbortingSequence +1;				
		END_IF
		
	21: IF ipMotionSystem.P_ResetMovers.Done THEN
			nAbortingSequence := nAbortingSequence +9;
		ELSIF ipMotionSystem.P_ResetMovers.Error THEN
			nAbortingSequence := nAbortingSequence +1;		
		END_IF

	22:	// Check error ID and react accordingly
		nErrorID := ipMotionSystem.P_ResetMovers.ErrorID;			
		ipVisuMessage.SetErrorMessage('RESET failed', 'Aborting', nAbortingSequence, nErrorID);			
		
		
	30: // Disable all movers	
		IF ipMotionSystem.DisableMovers() THEN
			ipVisuMessage.SetInfoMessage('DISABLE Movers', 'Aborting', nAbortingSequence);
			nAbortingSequence := nAbortingSequence +1;
		ELSE
			nAbortingSequence := nAbortingSequence +5;
		END_IF
		
	31: IF ipMotionSystem.P_DisableMovers.Done THEN
			nAbortingSequence := nAbortingSequence +9;
					
		ELSIF ipMotionSystem.P_DisableMovers.Error THEN
			nAbortingSequence := nAbortingSequence +1;					
		END_IF

	32:	// Check error ID and react accordingly
		nErrorID := ipMotionSystem.P_DisableMovers.ErrorID;	
		ipVisuMessage.SetErrorMessage('DISABLE failed', 'Aborting', nAbortingSequence, nErrorID);	
		
		
		
	40:	// Remove Tracks from Group
		IF ipMotionSystem.RemoveTracksFromGroup() THEN
			ipVisuMessage.SetInfoMessage('REMOVE TRACKS FROM GROUP', 'Aborting', nAbortingSequence);
			nAbortingSequence := nAbortingSequence +1;
		END_IF	

	41: IF ipMotionSystem.P_RemoveTracksFromGroup.Done THEN
			nAbortingSequence := nAbortingSequence +9;
		ELSIF ipMotionSystem.P_RemoveTracksFromGroup.Error THEN
			nAbortingSequence := nAbortingSequence +1;	
		END_IF
		
	42:	// Check error ID and react accordingly
		nErrorID := ipMotionSystem.P_RemoveTracksFromGroup.ErrorID;
		ipVisuMessage.SetErrorMessage('REMOVE TRACKS FROM GROUP failed', 'Aborting', nAbortingSequence, nErrorID);			
		
		
		
	50: // Remove Environment from Group
		IF ipMotionSystem.RemoveEnvironmentFromGroup() THEN
			ipVisuMessage.SetInfoMessage('REMOVE ENVIRONMENT FROM GROUP', 'Aborting', nAbortingSequence);
			nAbortingSequence := nAbortingSequence +1;
		END_IF	
		
	51: IF ipMotionSystem.P_RemoveEnviromentFromGroup.Done THEN
			nAbortingSequence := nAbortingSequence +9;
		ELSIF ipMotionSystem.P_RemoveEnviromentFromGroup.Error THEN
			nAbortingSequence := nAbortingSequence +1;				
		END_IF		

	52:	// Check error ID and react accordingly
		nErrorID := ipMotionSystem.P_RemoveEnviromentFromGroup.ErrorID;	
		ipVisuMessage.SetErrorMessage('REMOVE ENVIRONMENT FROM GROUP failed', 'Aborting', nAbortingSequence, nErrorID);			
		
		
		
	60: // Disable group
		IF ipMotionSystem.DisableGroup() THEN
			ipVisuMessage.SetInfoMessage('DISABLE GROUP', 'Aborting', nAbortingSequence);
			nAbortingSequence := nAbortingSequence +1;
		END_IF

	61: IF ipMotionSystem.P_DisableGroup.Done THEN
			nAbortingSequence := nAbortingSequence +9;
		ELSIF ipMotionSystem.P_DisableGroup.Error THEN
			nAbortingSequence := nAbortingSequence +1;					
		END_IF		
	
	62:	// Check error ID and react accordingly
		nErrorID := ipMotionSystem.P_DisableGroup.ErrorID;
		ipVisuMessage.SetErrorMessage('DISABLE GROUP failed', 'Aborting', nAbortingSequence, nErrorID);		


		
	70: // Disable all tracks
		IF ipMotionSystem.DisableTracks() THEN
			ipVisuMessage.SetInfoMessage('DISABLE TRACKS', 'Aborting', nAbortingSequence);
			nAbortingSequence := nAbortingSequence +1;
		END_IF
		
	71:	IF ipMotionSystem.P_DisableTracks.Done THEN
			nAbortingSequence := nAbortingSequence +9;
		ELSIF ipMotionSystem.P_DisableTracks.Error THEN
			nAbortingSequence := nAbortingSequence +1;
		END_IF
	
	72:	nErrorID := ipMotionSystem.P_DisableTracks.ErrorID;
		ipVisuMessage.SetErrorMessage('DISABLE TRACKS failed', 'Aborting', nAbortingSequence, nErrorID);	


	80:	nAbortingSequence := 100;


		
	100: // Reset of all sequences / Aborting done
		ipVisuMessage.SetInfoMessage('ABORTING finished', 'Aborting', 0);
	
		nAbortingSequence  := 0;
		nResettingSequence := 0;
		nPrepareSequence   := 0;
		nExecutingSequence := 0;
		          Aborting := TRUE;
				  
 		  
END_CASE


	ipVisuMessage.StateUpdate(nAbortingSequence, 'Aborting');
END_METHOD

METHOD Cycle : BOOL
VAR_INPUT
END_VAR


VAR_INST
	nMoverIndex	: UDINT;
	nTestCnt	: UINT;
END_VAR

	nTestCnt := nTestCnt +1;


	// Keeping the std cycle alive
	IF THIS^.std <> 0 THEN
		THIS^.std.Cycle();
	END_IF



	// Scanning for mover error e.g. Following Error
	bMoverError := FALSE;
	FOR nMoverIndex:=1 TO g_nMoverCount DO	
		IF ipMoverApplication[nMoverIndex] <> 0 THEN
			IF ipMoverApplication[nMoverIndex].std.P_State = MC_PLANAR_STATE.Error THEN
				bMoverError := TRUE;	
			END_IF
		END_IF
	END_FOR
END_METHOD

METHOD Execute : UDINT

	CASE nExecutingSequence OF
		
	
	0:	// Enter
		ipVisuMessage.ClearAllMessages();
		nExecutingSequence := 10;
	
	
	10: // Setting all stations into production mode
		FOR idx:=1 TO gc_NumberStations DO
			ipStation[idx].P_eProcessMode := E_ProcessMode.Production;
		END_FOR
		nExecutingSequence := 100;
		
		
		
	100: // Execution	
		;
	

	END_CASE
END_METHOD

METHOD MoverPreparation : BOOL
VAR_INPUT
	bReset 	: BOOL;
END_VAR


VAR_INST
	
	nStatePreparation		: DINT;
	
	
	operationMode				: XPlanarOperationMode; 
	
	idx2						: UDINT;

	nTileDcLinkVoltage			: UINT;
	bTilePowerOK				: BOOL;
	bTilePowerOverview			: ARRAY[1..gc_MaxNumberTiles] OF BOOL;
	bPowerOK					: BOOL;
	bPowerMissing				: BOOL;
	nTileCount					: UDINT;
	nTileToCheck				: UINT;
	bWithBumperID				: BOOL;	
	nMoverAccessoryIdCount		: ARRAY[1..gc_nMaxNumberMovers] OF UDINT;	
	
	stStartCheck 				: ST_CheckStartConditionFeedback;
	nLimitExceeded_MoverID		: UDINT;
	bLimitExceeded_Angle 		: BOOL;
	bLimitExceeded_PositionX 	: BOOL;
	bLimitExceeded_PositionY 	: BOOL;	
	fCurrentAngleDeviation		: LREAL;
	fCurrentPositionDeviationX	: LREAL;
	fCurrentPositionDeviationY	: LREAL;	

	sTextTemp					: STRING;

	eMoverAccessoryID			: MoverAccessoryID;

	
	moverCoordComStatus			: CoordinatedMoverCommStatus;
	moverComStatus				: MoverCommunicationStatus;
	
	bMoverCommunicationProblem  : ARRAY[1..gc_nMaxNumberMovers] OF BOOL;
	bCommunicationProblem		: BOOL;
	
	nMoverToCorrect				: UDINT;
	fMoverOrientationRead		: LREAL;
	fMoverOrientationCorrect	: LREAL;
	bDoRotationCorrection		: BOOL;
	CorrectionPos				: PositionXYC;
	
	bDeterminedMoverID				: BOOL;
	bDerterminedMoverOrientation 	: BOOL;
	
	fPosX							: LREAL;
	fPosY							: LREAL;
	fPosC							: LREAL;
	
	nCommunicationRetryCounter		: UINT;
	
	nMoverToCheck					: UINT;
	
	nMoverID_ErrorCode				: DWORD;
	
	MoverType						: XPlanarMoverType;
	bMoverCanDeterminOrientation	: BOOL;
END_VAR
IF bReset THEN
	nStatePreparation := 0;
	MoverPreparation := TRUE;
END_IF


	CASE nStatePreparation OF
		
	0:  nStatePreparation := 10;
	

	10: // 1st: Check if the system is in simulation mode or not
		// Simulation > OperationMode = 1
		//     Normal > OperationMode = 0
	    operationMode := ipMotionSystem.ipDriver.XpuTcIo(1).GetOperationMode();	
		IF operationMode = 0 THEN
			bPowerMissing := FALSE;
			nStatePreparation := nStatePreparation + 10;
		ELSE
			nStatePreparation := 500;
		END_IF
	
		
	20: // 2nd: Check power of each tile
		IF NOT bPowerMissing THEN
			ipVisuMessage.SetInfoMessage('Checking tile power', 'MoverPreparation', nStatePreparation);
		ELSE
			ipVisuMessage.SetErrorMessage('Tile power missing!', 'MoverPreparation', nStatePreparation, 0);	
		END_IF
		
		    bPowerOK := TRUE;
		nTileToCheck := 0;
		  nTileCount := ipMotionSystem.ipDriver.XpuTcIo(1).GetTileCount();
		
		nStatePreparation := nStatePreparation + 1;
		
	21:
		nTileToCheck := nTileToCheck +1;
		IF nTileToCheck <= nTileCount THEN
			nStatePreparation := nStatePreparation + 1;
		ELSE
			IF bPowerOK THEN
				nStatePreparation := nStatePreparation + 9;
			ELSE
				bPowerMissing := TRUE;
				nStatePreparation := nStatePreparation - 1;
			END_IF
		END_IF
		
	22:
		nTileDcLinkVoltage := ipMotionSystem.ipDriver.XpuTcIo(1).TileTcIo(1,nTileToCheck).GetActDcLinkVoltage(); 
		IF nTileDcLinkVoltage > 6000 THEN
			bTilePowerOK := TRUE;
		ELSE
			bTilePowerOK := FALSE;	
		END_IF
		bPowerOK := bPowerOK AND bTilePowerOK;
		bTilePowerOverview[nTileToCheck] := bPowerOK;
		nStatePreparation := nStatePreparation - 1;
		
		
		
	30:// 3rd: Mover re-detection, in case a mover was removed inbetween
	
		// Check if a mover has been lost...
		IF ipMotionSystem.CheckValidMovers() THEN
			ipVisuMessage.SetInfoMessage('Mover re-detection', 'MoverPreparation', nStatePreparation);
			nStatePreparation := nStatePreparation + 1;
		END_IF
	
	31:
		IF ipMotionSystem.P_CheckValidMovers.bDone THEN
			IF ipMotionSystem.P_CheckValidMovers.bMoverLost THEN
				         bDeterminedMoverID := FALSE;
				bDerterminedMoverOrientation := FALSE;
				nStatePreparation := nStatePreparation + 1;
			ELSE
				nStatePreparation := nStatePreparation + 9;
			END_IF
		END_IF
				
		bDeterminedMoverID := FALSE;
		bDerterminedMoverOrientation := FALSE;		
		
		
	32: // Starting mover re-detection
		IF ipMotionSystem.UtilityCheckForError(bAutoReset := TRUE) > 0 THEN
			IF ipMotionSystem.ipDriver.XpuTcIo(1).SetStartMoverRedetection() THEN	
				nStatePreparation := nStatePreparation +1;
			END_IF
		END_IF
	
	33: // Checking if all movers have been found on the XPlanar surface
		stMoverDetectionInfos := ipMotionSystem.ipDriver.XpuTcIo(1).GetMoverDetectionInfos();
		
		IF stMoverDetectionInfos.APM4220Detected = stMoverDetectionInfos.APM4220Expected THEN
			nStatePreparation := nStatePreparation +7;
		ELSE
			sTextTemp := 'Mover Missing!  Expected:';
			sTextTemp := CONCAT(sTextTemp, UDINT_TO_STRING(stMoverDetectionInfos.APM4220Detected));
			sTextTemp := CONCAT(sTextTemp, '  Detected:');
			sTextTemp := CONCAT(sTextTemp, UDINT_TO_STRING(stMoverDetectionInfos.APM4220Detected));
			
			ipVisuMessage.SetErrorMessage(sTextTemp, 'MoverPreparation', nStatePreparation, 0);	
		END_IF
	
		
	
	 40: // 4th: Checking the position of each mover before enabeling
	 	ipVisuMessage.SetInfoMessage('Check mover position', 'MoverPreparation', nStatePreparation);
	 
		bDone := TRUE;
		FOR idx:=1 TO g_nMoverCount DO
			stStartCheck := ipMoverApplication[idx].std.CheckStartConditions();
			IF NOT stStartCheck.bPositionOK THEN
				bDone := FALSE;
				EXIT;
			END_IF			
		END_FOR
	
		IF bDone THEN
			nStatePreparation := nStatePreparation + 2;
		ELSE
			nStatePreparation := nStatePreparation + 1;
		END_IF
			
	 41: // Position-Check failed:
		 // Except for rotation-points between four quadrants the angle limit of the c-axis is +/- 10.0°
		 // At rotation-points the max position deviation is +/-1mm in x/y-direction  	
				nLimitExceeded_MoverID := stStartCheck.nMoverID;
				  bLimitExceeded_Angle := stStartCheck.bAngleLimitExceeded;
			  bLimitExceeded_PositionX := stStartCheck.bPositionXLimitExceeded;
			  bLimitExceeded_PositionY := stStartCheck.bPositionYLimitExceeded;	
				fCurrentAngleDeviation := stStartCheck.fCurrentAngleDeviation;
			fCurrentPositionDeviationX := stStartCheck.fCurrentPositionDeviationX;
			fCurrentPositionDeviationY := stStartCheck.fCurrentPositionDeviationY;
	
			sTextTemp := 'Position Check Failed! - Mover ';
			sTextTemp := CONCAT(sTextTemp, UDINT_TO_STRING(nLimitExceeded_MoverID));
			sTextTemp := CONCAT(sTextTemp, ' too far away from rotation point.');
			
			ipVisuMessage.SetErrorMessage(sTextTemp, 'MoverPreparation', nStatePreparation, 0);	
			
			nStatePreparation := nStatePreparation - 1;
			
	42:		ipVisuMessage.ClearAllMessages();
			nStatePreparation := nStatePreparation + 8;
		
		
		
	50: // 5th: Check if movers with accessory MoverID are present. If yes, do mover identification before enabeling all movers.	
		bWithBumperID := FALSE;
			
		IF ipMotionSystem.UtilityCheckForError(bAutoReset := TRUE) > 0 THEN
			FOR idx:=1 TO g_nMoverCount DO
				nMoverAccessoryIdCount[idx] := ipMotionSystem.ipDriver.XpuTcIo(1).MoverTcIo(UDINT_TO_UINT(idx)).GetAccessoryIdCount();
			END_FOR
			
			FOR idx:=1 TO g_nMoverCount DO
				FOR idx2:=1 TO nMoverAccessoryIdCount[idx] DO
					eMoverAccessoryID := ipMotionSystem.ipDriver.XpuTcIo(1).MoverTcIo(UDINT_TO_UINT(idx)).GetAccessoryID(UDINT_TO_UINT(idx2));
					
					IF eMoverAccessoryID = MoverAccessoryID.APM9001_0000 THEN
						// Note: With the current driver release (3.2209.36.0) mover identification only works if all movers are equiped with ID bumpers!
						bWithBumperID := TRUE;						
					END_IF
				END_FOR
			END_FOR
		END_IF

			
		IF bWithBumperID THEN
			nStatePreparation := nStatePreparation + 10;
		ELSE
			nStatePreparation := 500;
		END_IF
		
		
	60: // 6th: Do mover identification
		ipVisuMessage.SetInfoMessage('Start mover-identification', 'MoverPreparation', nStatePreparation);
	
		IF NOT bDeterminedMoverID THEN
			IF ipMotionSystem.UtilityCheckForError(bAutoReset := TRUE) > 0 THEN
				IF ipMotionSystem.ipDriver.XpuTcIo(1).SetCoordMoverCommunicationCmd(CoordinatedMoverCommCommand.IdentifyAndAssignPossible) THEN
					nStatePreparation := nStatePreparation +1;
				END_IF	
			END_IF
		ELSE
			nStatePreparation := nStatePreparation +10;
		END_IF
	
	61:
		IF ipMotionSystem.UtilityCheckForError(bAutoReset := TRUE) > 0 THEN			
			moverCoordComStatus := ipMotionSystem.ipDriver.XpuTcIo(1).GetCoordMoverCommStatus();
			
			IF moverCoordComStatus = CoordinatedMoverCommStatus.CommunicationSuccessful THEN
				bDeterminedMoverID := TRUE;
				ipVisuMessage.ClearAllMessages();
				nStatePreparation := nStatePreparation + 9;	
			ELSIF moverCoordComStatus = CoordinatedMoverCommStatus.CommunicationFailed THEN
				nStatePreparation := nStatePreparation + 1;	
			END_IF
			
		END_IF
		
	62:	IF ipMotionSystem.UtilityCheckForError(bAutoReset := TRUE) > 0 THEN	
			nMoverID_ErrorCode := ipMotionSystem.ipDriver.XpuTcIo(1).GetCoordMoverCommunicationErrorId();
			ipVisuMessage.SetErrorMessage('Mover Identification Failed!', 'MoverPreparation', nStatePreparation, nMoverID_ErrorCode);
		END_IF
		
		IF ipVisuMessage.CheckAknowledge()  THEN
			nStatePreparation := 0;	
		END_IF
		
		
		
	70: // 7th: Determine Mover-Orientation
	
		// Note: At the time of creation of this example code only APM4330 was able to determine its orientation.
		//       Change the code according to newer driver releases and availability of the orientation feature.
		bMoverCanDeterminOrientation := TRUE;
		FOR idx:=1 TO g_nMoverCount DO
			MoverType := ipMotionSystem.ipDriver.XpuTcIo(1).MoverTcIo(UDINT_TO_UINT(idx)).GetMoverType();
			IF MoverType <> XPlanarMoverType.APM4330 THEN
				bMoverCanDeterminOrientation := FALSE;
			END_IF
		END_FOR
			
		IF bMoverCanDeterminOrientation THEN
			IF NOT bDerterminedMoverOrientation THEN
				ipVisuMessage.SetInfoMessage('Mover orientation determination', 'MoverPreparation', nStatePreparation);
				IF ipMotionSystem.UtilityCheckForError(bAutoReset := TRUE) > 0 THEN
					IF ipMotionSystem.ipDriver.XpuTcIo(1).SetCoordMoverCommunicationCmd(CoordinatedMoverCommCommand.DetermineOrientations) THEN
						nStatePreparation := nStatePreparation + 1;	
					END_IF
				END_IF
			ELSE
				nStatePreparation := nStatePreparation + 20;		
			END_IF
		ELSE
			nStatePreparation := nStatePreparation + 20;
		END_IF
	
		
	71: // Check if communication is active
		IF ipMotionSystem.UtilityCheckForError(bAutoReset := TRUE) > 0 THEN
			moverCoordComStatus := ipMotionSystem.ipDriver.XpuTcIo(1).GetCoordMoverCommStatus();
			IF moverCoordComStatus = CoordinatedMoverCommStatus.CommunicationInProcess THEN
				nStatePreparation := nStatePreparation + 1;	
			END_IF
		END_IF
	
		
	72: // Wait for orientation determination finished
		IF ipMotionSystem.UtilityCheckForError(bAutoReset := TRUE) > 0 THEN
			moverCoordComStatus := ipMotionSystem.ipDriver.XpuTcIo(1).GetCoordMoverCommStatus();
			IF moverCoordComStatus = CoordinatedMoverCommStatus.CommunicationSuccessful THEN
				nStatePreparation := nStatePreparation + 8;	
			ELSIF moverCoordComStatus = CoordinatedMoverCommStatus.CommunicationFailed THEN
				IF nCommunicationRetryCounter <= 5 THEN
					nCommunicationRetryCounter := nCommunicationRetryCounter +1;
					nStatePreparation := nStatePreparation - 2;	
				ELSE
					nStatePreparation := nStatePreparation + 1;	
				END_IF
			END_IF
		END_IF
		
				
	73:	// Check which movers do not communicate correctly:
		nMoverToCheck := 0;
		nStatePreparation := nStatePreparation + 1;
		
	74: nMoverToCheck := nMoverToCheck +1;
		IF nMoverToCheck <= g_nMoverCount THEN
			IF ipMotionSystem.UtilityCheckForError(bAutoReset := TRUE) > 0 THEN
				IF ipMotionSystem.ipDriver.XpuTcIo(1).MoverTcIo(nMoverToCheck).SetMoverCommunicationCommand(MoverCommunicationCommand.DetermineOrientation) THEN
					nStatePreparation := nStatePreparation + 1;
				END_IF
			END_IF
		ELSE
			FOR idx:=1 TO g_nMoverCount DO
				bCommunicationProblem := FALSE;
				IF bMoverCommunicationProblem[idx] THEN
					bCommunicationProblem := TRUE;	
				END_IF
			END_FOR
			
			IF bCommunicationProblem THEN
				sTextTemp := 'Mover Communication Problem: ';
				FOR idx:=1 TO g_nMoverCount DO
					IF bMoverCommunicationProblem[idx] THEN
						sTextTemp := CONCAT(sTextTemp, ' M');
						sTextTemp := CONCAT(sTextTemp, UDINT_TO_STRING(idx));
					END_IF
				END_FOR				
				ipVisuMessage.SetErrorMessage(sTextTemp, sTextTemp, nStatePreparation, 0);
			ELSE
				nStatePreparation := nStatePreparation - 4;	
			END_IF
		END_IF
		
	75: moverComStatus := ipMotionSystem.ipDriver.XpuTcIo(1).MoverTcIo(nMoverToCheck).GetCommunicationStatus();
		IF moverComStatus = MoverCommunicationStatus.CommunicationSuccessful THEN
			bMoverCommunicationProblem[nMoverToCheck] := FALSE;
			nStatePreparation := nStatePreparation - 1;
		ELSIF moverComStatus = MoverCommunicationStatus.CommunicationFailed THEN
			bMoverCommunicationProblem[nMoverToCheck] := TRUE;
			nStatePreparation := nStatePreparation - 1;
		END_IF
		
		
	80:	// Rotation-Angle modulo adaption
		ipVisuMessage.SetInfoMessage('Rotation-Angle modulo adaption', 'MoverPreparation', nStatePreparation);
		nMoverToCorrect := 0;
		nStatePreparation := nStatePreparation + 1;	
		
